KUKA KRL program: bl_1.src

&ACCESS RVP
&REL 1
&PARAM TEMPLATE = C:\KRC\Roboter\Template\vorgabe
&PARAM EDITMASK = *
DEF group15cm ( )


;FOLD INI
;FOLD BASISTECH INI
GLOBAL INTERRUPT DECL 3 WHEN $STOPMESS==TRUE DO IR_STOPM ( )
INTERRUPT ON 3
BAS (#INITMOV,0 )
;ENDFOLD (BASISTECH INI)
;ENDFOLD (INI)

;FOLD STARTPOSITION - BASE IS 2, TOOL IS 6, SPEED IS 45%, POSITION IS A1 5,A2 -30,A3 100,A4 5,A5 -60,A6 -135,E1 0,E2 0,E3 0,E4 0
$BWDSTART = FALSE
PDAT_ACT = {VEL 45,ACC 100,APO_DIST 50}
FDAT_ACT = {TOOL_NO 6,BASE_NO 2,IPO_FRAME #BASE}
BAS (#PTP_PARAMS,45)
PTP  {A1 5,A2 -30,A3 100,A4 5,A5 -60,A6 -135,E1 0,E2 0,E3 0,E4 0}
;ENDFOLD

;FOLD LIN SPEED IS 0.5 m/sec, INTERPOLATION SETTINGS IN FOLD
$VEL.CP=0.5
$ADVANCE=3
;ENDFOLD

PTP{ E6POS: X 793.0310, Y -5.4900, Z -174.0150, A 0, B 90, C 0, E1 0, E2 0, E3 0, E4 0, S 'B 110' } C_PTP
LIN{ E6POS: X 793.0310, Y -5.4900, Z -174.0150, A 0, B 90, C 0, E1 0, E2 0, E3 0, E4 0 }
LIN{ E6POS: X 792.7476, Y -6.4490, Z -174.0150, A 0, B 90, C 0, E1 0, E2 0, E3 0, E4 0 } C_DIS
LIN{ E6POS: X 792.4642, Y -7.4080, Z -174.0150, A 0, B 90, C 0, E1 0, E2 0, E3 0, E4 0 } C_DIS
LIN{ E6POS: X 792.1808, Y -8.3670, Z -174.0150, A 0, B 90, C 0, E1 0, E2 0, E3 0, E4 0 } C_DIS
LIN{ E6POS: X 791.8974, Y -9.3260, Z -174.0150, A 0, B 90, C 0, E1 0, E2 0, E3 0, E4 0 } C_DIS
LIN{ E6POS: X 791.6139, Y -10.2850, Z -174.0150, A 0, B 90, C 0, E1 0, E2 0, E3 0, E4 0 } C_DIS
LIN{ E6POS: X 791.3305, Y -11.2440, Z -174.0150, A 0, B 90, C 0, E1 0, E2 0, E3 0, E4 0 } C_DIS
LIN{ E6POS: X 791.0471, Y -12.2030, Z -174.0150, A 0, B 90, C 0, E1 0, E2 0, E3 0, E4 0 } C_DIS
LIN{ E6POS: X 790.7637, Y -13.1620, Z -174.0150, A 0, B 90, C 0, E1 0, E2 0, E3 0, E4 0 } C_DIS
LIN{ E6POS: X 790.4803, Y -14.1210, Z -174.0150, A 0, B 90, C 0, E1 0, E2 0, E3 0, E4 0 } C_DIS
LIN{ E6POS: X 790.2681, Y -14.8387, Z -174.0150, A 0, B 90, C 0, E1 0, E2 0, E3 0, E4 0 } C_DIS
LIN{ E6POS: X 790.2681, Y -14.8387, Z -174.0150, A 0, B 90, C 0, E1 0, E2 0, E3 0, E4 0 } C_DIS
LIN{ E6POS: X 789.6733, Y -15.6426, Z -174.0150, A 0, B 90, C 0, E1 0, E2 0, E3 0, E4 0 } C_DIS
LIN{ E6POS: X 789.0784, Y -16.4464, Z -174.0150, A 0, B 90, C 0, E1 0, E2 0, E3 0, E4 0 } C_DIS
LIN{ E6POS: X 788.4835, Y -17.2502, Z -174.0150, A 0, B 90, C 0, E1 0, E2 0, E3 0, E4 0 } C_DIS
LIN{ E6POS: X 787.8887, Y -18.0540, Z -174.0150, A 0, B 90, C 0, E1 0, E2 0, E3 0, E4 0 } C_DIS
LIN{ E6POS: X 787.2938, Y -18.8579, Z -174.0150, A 0, B 90, C 0, E1 0, E2 0, E3 0, E4 0 } C_DIS
LIN{ E6POS: X 786.7884, Y -19.5408, Z -174.0150, A 0, B 90, C 0, E1 0, E2 0, E3 0, E4 0 } C_DIS
LIN{ E6POS: X 786.7884, Y -19.5408, Z -174.0150, A 0, B 90, C 0, E1 0, E2 0, E3 0, E4 0 } C_DIS
LIN{ E6POS: X 785.8349, Y -19.8419, Z -174.0150, A 0, B 90, C 0, E1 0, E2 0, E3 0, E4 0 } C_DIS
LIN{ E6POS: X 784.8813, Y -20.1431, Z -174.0150, A 0, B 90, C 0, E1 0, E2 0, E3 0, E4 0 } C_DIS
LIN{ E6POS: X 783.9277, Y -20.4443, Z -174.0150, A 0, B 90, C 0, E1 0, E2 0, E3 0, E4 0 } C_DIS
LIN{ E6POS: X 782.9742, Y -20.7455, Z -174.0150, A 0, B 90, C 0, E1 0, E2 0, E3 0, E4 0 } C_DIS
LIN{ E6POS: X 782.5387, Y -20.8830, Z -174.0150, A 0, B 90, C 0, E1 0, E2 0, E3 0, E4 0 } C_DIS
LIN{ E6POS: X 781.5488, Y -20.7411, Z -174.0150, A 0, B 90, C 0, E1 0, E2 0, E3 0, E4 0 } C_DIS
LIN{ E6POS: X 780.5590, Y -20.5992, Z -174.0150, A 0, B 90, C 0, E1 0, E2 0, E3 0, E4 0 } C_DIS
LIN{ E6POS: X 779.5691, Y -20.4573, Z -174.0150, A 0, B 90, C 0, E1 0, E2 0, E3 0, E4 0 } C_DIS
LIN{ E6POS: X 778.5792, Y -20.3154, Z -174.0150, A 0, B 90, C 0, E1 0, E2 0, E3 0, E4 0 } C_DIS
LIN{ E6POS: X 777.5893, Y -20.1735, Z -174.0150, A 0, B 90, C 0, E1 0, E2 0, E3 0, E4 0 } C_DIS
LIN{ E6POS: X 777.4677, Y -20.1560, Z -174.0150, A 0, B 90, C 0, E1 0, E2 0, E3 0, E4 0 } C_DIS
LIN{ E6POS: X 777.4677, Y -20.1560, Z -174.0150, A 0, B 90, C 0, E1 0, E2 0, E3 0, E4 0 } C_DIS
LIN{ E6POS: X 776.4984, Y -19.9101, Z -174.0150, A 0, B 90, C 0, E1 0, E2 0, E3 0, E4 0 } C_DIS
LIN{ E6POS: X 775.5291, Y -19.6643, Z -174.0150, A 0, B 90, C 0, E1 0, E2 0, E3 0, E4 0 } C_DIS
LIN{ E6POS: X 774.5598, Y -19.4184, Z -174.0150, A 0, B 90, C 0, E1 0, E2 0, E3 0, E4 0 } C_DIS
LIN{ E6POS: X 773.5905, Y -19.1725, Z -174.0150, A 0, B 90, C 0, E1 0, E2 0, E3 0, E4 0 } C_DIS
LIN{ E6POS: X 772.6212, Y -18.9266, Z -174.0150, A 0, B 90, C 0, E1 0, E2 0, E3 0, E4 0 } C_DIS
LIN{ E6POS: X 771.6519, Y -18.6807, Z -174.0150, A 0, B 90, C 0, E1 0, E2 0, E3 0, E4 0 } C_DIS
LIN{ E6POS: X 771.5220, Y -18.6477, Z -174.0150, A 0, B 90, C 0, E1 0, E2 0, E3 0, E4 0 } C_DIS
LIN{ E6POS: X 771.5220, Y -18.6477, Z -174.0150, A 0, B 90, C 0, E1 0, E2 0, E3 0, E4 0 } C_DIS
LIN{ E6POS: X 770.5324, Y -18.5039, Z -174.0150, A 0, B 90, C 0, E1 0, E2 0, E3 0, E4 0 } C_DIS
LIN{ E6POS: X 769.5428, Y -18.3600, Z -174.0150, A 0, B 90, C 0, E1 0, E2 0, E3 0, E4 0 } C_DIS
LIN{ E6POS: X 768.5532, Y -18.2161, Z -174.0150, A 0, B 90, C 0, E1 0, E2 0, E3 0, E4 0 } C_DIS
LIN{ E6POS: X 767.5636, Y -18.0723, Z -174.0150, A 0, B 90, C 0, E1 0, E2 0, E3 0, E4 0 } C_DIS
LIN{ E6POS: X 766.5740, Y -17.9284, Z -174.0150, A 0, B 90, C 0, E1 0, E2 0, E3 0, E4 0 } C_DIS
LIN{ E6POS: X 765.5844, Y -17.7845, Z -174.0150, A 0, B 90, C 0, E1 0, E2 0, E3 0, E4 0 } C_DIS
LIN{ E6POS: X 764.6502, Y -17.6487, Z -174.0150, A 0, B 90, C 0, E1 0, E2 0, E3 0, E4 0 } C_DIS
LIN{ E6POS: X 764.6502, Y -17.6487, Z -174.0150, A 0, B 90, C 0, E1 0, E2 0, E3 0, E4 0 } C_DIS
LIN{ E6POS: X 763.6529, Y -17.5756, Z -174.0150, A 0, B 90, C 0, E1 0, E2 0, E3 0, E4 0 } C_DIS
LIN{ E6POS: X 762.6555, Y -17.5025, Z -174.0150, A 0, B 90, C 0, E1 0, E2 0, E3 0, E4 0 } C_DIS
LIN{ E6POS: X 761.6582, Y -17.4294, Z -174.0150, A 0, B 90, C 0, E1 0, E2 0, E3 0, E4 0 } C_DIS
LIN{ E6POS: X 760.6609, Y -17.3562, Z -174.0150, A 0, B 90, C 0, E1 0, E2 0, E3 0, E4 0 } C_DIS
LIN{ E6POS: X 759.6636, Y -17.2831, Z -174.0150, A 0, B 90, C 0, E1 0, E2 0, E3 0, E4 0 } C_DIS
LIN{ E6POS: X 758.6662, Y -17.2100, Z -174.0150, A 0, B 90, C 0, E1 0, E2 0, E3 0, E4 0 } C_DIS
LIN{ E6POS: X 757.6689, Y -17.1369, Z -174.0150, A 0, B 90, C 0, E1 0, E2 0, E3 0, E4 0 } C_DIS
LIN{ E6POS: X 757.5979, Y -17.1316, Z -174.0150, A 0, B 90, C 0, E1 0, E2 0, E3 0, E4 0 } C_DIS
LIN{ E6POS: X 757.5979, Y -17.1316, Z -174.0150, A 0, B 90, C 0, E1 0, E2 0, E3 0, E4 0 } C_DIS
LIN{ E6POS: X 756.5980, Y -17.1225, Z -174.0150, A 0, B 90, C 0, E1 0, E2 0, E3 0, E4 0 } C_DIS
LIN{ E6POS: X 755.5980, Y -17.1134, Z -174.0150, A 0, B 90, C 0, E1 0, E2 0, E3 0, E4 0 } C_DIS
LIN{ E6POS: X 754.5981, Y -17.1043, Z -174.0150, A 0, B 90, C 0, E1 0, E2 0, E3 0, E4 0 } C_DIS
LIN{ E6POS: X 753.5981, Y -17.0952, Z -174.0150, A 0, B 90, C 0, E1 0, E2 0, E3 0, E4 0 } C_DIS
LIN{ E6POS: X 752.5981, Y -17.0860, Z -174.0150, A 0, B 90, C 0, E1 0, E2 0, E3 0, E4 0 } C_DIS
LIN{ E6POS: X 751.5982, Y -17.0769, Z -174.0150, A 0, B 90, C 0, E1 0, E2 0, E3 0, E4 0 } C_DIS
LIN{ E6POS: X 751.1080, Y -17.0724, Z -174.0150, A 0, B 90, C 0, E1 0, E2 0, E3 0, E4 0 } C_DIS
LIN{ E6POS: X 751.1080, Y -17.0724, Z -174.0150, A 0, B 90, C 0, E1 0, E2 0, E3 0, E4 0 } C_DIS
LIN{ E6POS: X 750.1105, Y -17.1440, Z -174.0150, A 0, B 90, C 0, E1 0, E2 0, E3 0, E4 0 } C_DIS
LIN{ E6POS: X 749.1131, Y -17.2155, Z -174.0150, A 0, B 90, C 0, E1 0, E2 0, E3 0, E4 0 } C_DIS
LIN{ E6POS: X 748.1157, Y -17.2870, Z -174.0150, A 0, B 90, C 0, E1 0, E2 0, E3 0, E4 0 } C_DIS
LIN{ E6POS: X 747.1182, Y -17.3586, Z -174.0150, A 0, B 90, C 0, E1 0, E2 0, E3 0, E4 0 } C_DIS
LIN{ E6POS: X 746.1208, Y -17.4301, Z -174.0150, A 0, B 90, C 0, E1 0, E2 0, E3 0, E4 0 } C_DIS
LIN{ E6POS: X 745.9267, Y -17.4440, Z -174.0150, A 0, B 90, C 0, E1 0, E2 0, E3 0, E4 0 } C_DIS
LIN{ E6POS: X 745.9267, Y -17.4440, Z -174.0150, A 0, B 90, C 0, E1 0, E2 0, E3 0, E4 0 } C_DIS
LIN{ E6POS: X 744.9564, Y -17.6858, Z -174.0150, A 0, B 90, C 0, E1 0, E2 0, E3 0, E4 0 } C_DIS
LIN{ E6POS: X 743.9861, Y -17.9276, Z -174.0150, A 0, B 90, C 0, E1 0, E2 0, E3 0, E4 0 } C_DIS
LIN{ E6POS: X 743.0157, Y -18.1693, Z -174.0150, A 0, B 90, C 0, E1 0, E2 0, E3 0, E4 0 } C_DIS
LIN{ E6POS: X 742.7996, Y -18.2232, Z -174.0150, A 0, B 90, C 0, E1 0, E2 0, E3 0, E4 0 } C_DIS
LIN{ E6POS: X 742.7996, Y -18.2232, Z -174.0150, A 0, B 90, C 0, E1 0, E2 0, E3 0, E4 0 } C_DIS
LIN{ E6POS: X 742.1156, Y -18.9526, Z -174.0150, A 0, B 90, C 0, E1 0, E2 0, E3 0, E4 0 } C_DIS
LIN{ E6POS: X 741.7327, Y -19.3609, Z -174.0150, A 0, B 90, C 0, E1 0, E2 0, E3 0, E4 0 } C_DIS
LIN{ E6POS: X 741.7327, Y -19.3609, Z -174.0150, A 0, B 90, C 0, E1 0, E2 0, E3 0, E4 0 } C_DIS
LIN{ E6POS: X 741.7327, Y -19.3609, Z -174.0150, A 0, B 90, C 0, E1 0, E2 0, E3 0, E4 0 } C_DIS
LIN{ E6POS: X 742.3016, Y -20.1832, Z -174.0150, A 0, B 90, C 0, E1 0, E2 0, E3 0, E4 0 } C_DIS
LIN{ E6POS: X 742.7345, Y -20.8088, Z -174.0150, A 0, B 90, C 0, E1 0, E2 0, E3 0, E4 0 } C_DIS
LIN{ E6POS: X 742.7345, Y -20.8088, Z -174.0150, A 0, B 90, C 0, E1 0, E2 0, E3 0, E4 0 } C_DIS
LIN{ E6POS: X 743.6084, Y -21.2949, Z -174.0150, A 0, B 90, C 0, E1 0, E2 0, E3 0, E4 0 } C_DIS
LIN{ E6POS: X 744.4823, Y -21.7810, Z -174.0150, A 0, B 90, C 0, E1 0, E2 0, E3 0, E4 0 } C_DIS
LIN{ E6POS: X 745.3563, Y -22.2671, Z -174.0150, A 0, B 90, C 0, E1 0, E2 0, E3 0, E4 0 } C_DIS
LIN{ E6POS: X 745.8115, Y -22.5203, Z -174.0150, A 0, B 90, C 0, E1 0, E2 0, E3 0, E4 0 } C_DIS
LIN{ E6POS: X 745.8115, Y -22.5203, Z -174.0150, A 0, B 90, C 0, E1 0, E2 0, E3 0, E4 0 } C_DIS
LIN{ E6POS: X 746.7484, Y -22.8698, Z -174.0150, A 0, B 90, C 0, E1 0, E2 0, E3 0, E4 0 } C_DIS
LIN{ E6POS: X 747.6853, Y -23.2194, Z -174.0150, A 0, B 90, C 0, E1 0, E2 0, E3 0, E4 0 } C_DIS
LIN{ E6POS: X 748.6222, Y -23.5690, Z -174.0150, A 0, B 90, C 0, E1 0, E2 0, E3 0, E4 0 } C_DIS
LIN{ E6POS: X 749.5592, Y -23.9186, Z -174.0150, A 0, B 90, C 0, E1 0, E2 0, E3 0, E4 0 } C_DIS
LIN{ E6POS: X 750.4961, Y -24.2681, Z -174.0150, A 0, B 90, C 0, E1 0, E2 0, E3 0, E4 0 } C_DIS
LIN{ E6POS: X 750.9726, Y -24.4459, Z -174.0150, A 0, B 90, C 0, E1 0, E2 0, E3 0, E4 0 } C_DIS
LIN{ E6POS: X 750.9726, Y -24.4459, Z -174.0150, A 0, B 90, C 0, E1 0, E2 0, E3 0, E4 0 } C_DIS
LIN{ E6POS: X 751.9333, Y -24.7235, Z -174.0150, A 0, B 90, C 0, E1 0, E2 0, E3 0, E4 0 } C_DIS
LIN{ E6POS: X 752.8940, Y -25.0011, Z -174.0150, A 0, B 90, C 0, E1 0, E2 0, E3 0, E4 0 } C_DIS
LIN{ E6POS: X 753.8547, Y -25.2787, Z -174.0150, A 0, B 90, C 0, E1 0, E2 0, E3 0, E4 0 } C_DIS
LIN{ E6POS: X 754.8154, Y -25.5563, Z -174.0150, A 0, B 90, C 0, E1 0, E2 0, E3 0, E4 0 } C_DIS
LIN{ E6POS: X 755.7761, Y -25.8339, Z -174.0150, A 0, B 90, C 0, E1 0, E2 0, E3 0, E4 0 } C_DIS
LIN{ E6POS: X 756.7368, Y -26.1115, Z -174.0150, A 0, B 90, C 0, E1 0, E2 0, E3 0, E4 0 } C_DIS
LIN{ E6POS: X 757.4643, Y -26.3217, Z -174.0150, A 0, B 90, C 0, E1 0, E2 0, E3 0, E4 0 } C_DIS
LIN{ E6POS: X 757.4643, Y -26.3217, Z -174.0150, A 0, B 90, C 0, E1 0, E2 0, E3 0, E4 0 } C_DIS
LIN{ E6POS: X 758.4408, Y -26.5375, Z -174.0150, A 0, B 90, C 0, E1 0, E2 0, E3 0, E4 0 } C_DIS
LIN{ E6POS: X 759.4172, Y -26.7532, Z -174.0150, A 0, B 90, C 0, E1 0, E2 0, E3 0, E4 0 } C_DIS
LIN{ E6POS: X 760.3937, Y -26.9690, Z -174.0150, A 0, B 90, C 0, E1 0, E2 0, E3 0, E4 0 } C_DIS
LIN{ E6POS: X 761.3701, Y -27.1847, Z -174.0150, A 0, B 90, C 0, E1 0, E2 0, E3 0, E4 0 } C_DIS
LIN{ E6POS: X 762.3466, Y -27.4005, Z -174.0150, A 0, B 90, C 0, E1 0, E2 0, E3 0, E4 0 } C_DIS
LIN{ E6POS: X 763.3230, Y -27.6162, Z -174.0150, A 0, B 90, C 0, E1 0, E2 0, E3 0, E4 0 } C_DIS
LIN{ E6POS: X 764.2995, Y -27.8320, Z -174.0150, A 0, B 90, C 0, E1 0, E2 0, E3 0, E4 0 } C_DIS
LIN{ E6POS: X 764.5341, Y -27.8838, Z -174.0150, A 0, B 90, C 0, E1 0, E2 0, E3 0, E4 0 } C_DIS
LIN{ E6POS: X 764.5341, Y -27.8838, Z -174.0150, A 0, B 90, C 0, E1 0, E2 0, E3 0, E4 0 } C_DIS
LIN{ E6POS: X 765.5242, Y -28.0248, Z -174.0150, A 0, B 90, C 0, E1 0, E2 0, E3 0, E4 0 } C_DIS
LIN{ E6POS: X 766.5142, Y -28.1657, Z -174.0150, A 0, B 90, C 0, E1 0, E2 0, E3 0, E4 0 } C_DIS
LIN{ E6POS: X 767.5042, Y -28.3066, Z -174.0150, A 0, B 90, C 0, E1 0, E2 0, E3 0, E4 0 } C_DIS
LIN{ E6POS: X 768.4942, Y -28.4476, Z -174.0150, A 0, B 90, C 0, E1 0, E2 0, E3 0, E4 0 } C_DIS
LIN{ E6POS: X 769.4842, Y -28.5885, Z -174.0150, A 0, B 90, C 0, E1 0, E2 0, E3 0, E4 0 } C_DIS
LIN{ E6POS: X 770.4743, Y -28.7294, Z -174.0150, A 0, B 90, C 0, E1 0, E2 0, E3 0, E4 0 } C_DIS
LIN{ E6POS: X 771.4301, Y -28.8655, Z -174.0150, A 0, B 90, C 0, E1 0, E2 0, E3 0, E4 0 } C_DIS
LIN{ E6POS: X 771.4301, Y -28.8655, Z -174.0150, A 0, B 90, C 0, E1 0, E2 0, E3 0, E4 0 } C_DIS
LIN{ E6POS: X 772.4299, Y -28.8885, Z -174.0150, A 0, B 90, C 0, E1 0, E2 0, E3 0, E4 0 } C_DIS
LIN{ E6POS: X 773.4296, Y -28.9114, Z -174.0150, A 0, B 90, C 0, E1 0, E2 0, E3 0, E4 0 } C_DIS
LIN{ E6POS: X 774.4294, Y -28.9344, Z -174.0150, A 0, B 90, C 0, E1 0, E2 0, E3 0, E4 0 } C_DIS
LIN{ E6POS: X 775.4291, Y -28.9574, Z -174.0150, A 0, B 90, C 0, E1 0, E2 0, E3 0, E4 0 } C_DIS
LIN{ E6POS: X 776.4288, Y -28.9803, Z -174.0150, A 0, B 90, C 0, E1 0, E2 0, E3 0, E4 0 } C_DIS
LIN{ E6POS: X 777.3989, Y -29.0026, Z -174.0150, A 0, B 90, C 0, E1 0, E2 0, E3 0, E4 0 } C_DIS
LIN{ E6POS: X 777.3989, Y -29.0026, Z -174.0150, A 0, B 90, C 0, E1 0, E2 0, E3 0, E4 0 } C_DIS
LIN{ E6POS: X 778.3804, Y -29.1940, Z -174.0150, A 0, B 90, C 0, E1 0, E2 0, E3 0, E4 0 } C_DIS
LIN{ E6POS: X 779.3620, Y -29.3854, Z -174.0150, A 0, B 90, C 0, E1 0, E2 0, E3 0, E4 0 } C_DIS
LIN{ E6POS: X 780.3435, Y -29.5769, Z -174.0150, A 0, B 90, C 0, E1 0, E2 0, E3 0, E4 0 } C_DIS
LIN{ E6POS: X 781.3250, Y -29.7683, Z -174.0150, A 0, B 90, C 0, E1 0, E2 0, E3 0, E4 0 } C_DIS
LIN{ E6POS: X 782.0838, Y -29.9163, Z -174.0150, A 0, B 90, C 0, E1 0, E2 0, E3 0, E4 0 } C_DIS
LIN{ E6POS: X 782.0838, Y -29.9163, Z -174.0150, A 0, B 90, C 0, E1 0, E2 0, E3 0, E4 0 } C_DIS
LIN{ E6POS: X 782.7607, Y -30.6523, Z -174.0150, A 0, B 90, C 0, E1 0, E2 0, E3 0, E4 0 } C_DIS
LIN{ E6POS: X 783.4376, Y -31.3884, Z -174.0150, A 0, B 90, C 0, E1 0, E2 0, E3 0, E4 0 } C_DIS
LIN{ E6POS: X 784.1145, Y -32.1244, Z -174.0150, A 0, B 90, C 0, E1 0, E2 0, E3 0, E4 0 } C_DIS
LIN{ E6POS: X 784.7914, Y -32.8605, Z -174.0150, A 0, B 90, C 0, E1 0, E2 0, E3 0, E4 0 } C_DIS
LIN{ E6POS: X 785.1281, Y -33.2266, Z -174.0150, A 0, B 90, C 0, E1 0, E2 0, E3 0, E4 0 } C_DIS
LIN{ E6POS: X 785.1281, Y -33.2266, Z -174.0150, A 0, B 90, C 0, E1 0, E2 0, E3 0, E4 0 } C_DIS
LIN{ E6POS: X 785.2695, Y -34.2166, Z -174.0150, A 0, B 90, C 0, E1 0, E2 0, E3 0, E4 0 } C_DIS
LIN{ E6POS: X 785.4109, Y -35.2065, Z -174.0150, A 0, B 90, C 0, E1 0, E2 0, E3 0, E4 0 } C_DIS
LIN{ E6POS: X 785.5523, Y -36.1965, Z -174.0150, A 0, B 90, C 0, E1 0, E2 0, E3 0, E4 0 } C_DIS
LIN{ E6POS: X 785.6937, Y -37.1864, Z -174.0150, A 0, B 90, C 0, E1 0, E2 0, E3 0, E4 0 } C_DIS
LIN{ E6POS: X 785.8351, Y -38.1764, Z -174.0150, A 0, B 90, C 0, E1 0, E2 0, E3 0, E4 0 } C_DIS
LIN{ E6POS: X 785.9765, Y -39.1663, Z -174.0150, A 0, B 90, C 0, E1 0, E2 0, E3 0, E4 0 } C_DIS
LIN{ E6POS: X 786.1179, Y -40.1563, Z -174.0150, A 0, B 90, C 0, E1 0, E2 0, E3 0, E4 0 } C_DIS
LIN{ E6POS: X 786.1747, Y -40.5536, Z -174.0150, A 0, B 90, C 0, E1 0, E2 0, E3 0, E4 0 } C_DIS
LIN{ E6POS: X 786.1747, Y -40.5536, Z -174.0150, A 0, B 90, C 0, E1 0, E2 0, E3 0, E4 0 } C_DIS
LIN{ E6POS: X 786.0743, Y -41.5485, Z -174.0150, A 0, B 90, C 0, E1 0, E2 0, E3 0, E4 0 } C_DIS
LIN{ E6POS: X 785.9740, Y -42.5435, Z -174.0150, A 0, B 90, C 0, E1 0, E2 0, E3 0, E4 0 } C_DIS
LIN{ E6POS: X 785.8737, Y -43.5384, Z -174.0150, A 0, B 90, C 0, E1 0, E2 0, E3 0, E4 0 } C_DIS
LIN{ E6POS: X 785.7734, Y -44.5334, Z -174.0150, A 0, B 90, C 0, E1 0, E2 0, E3 0, E4 0 } C_DIS
LIN{ E6POS: X 785.6731, Y -45.5283, Z -174.0150, A 0, B 90, C 0, E1 0, E2 0, E3 0, E4 0 } C_DIS
LIN{ E6POS: X 785.5728, Y -46.5233, Z -174.0150, A 0, B 90, C 0, E1 0, E2 0, E3 0, E4 0 } C_DIS
LIN{ E6POS: X 785.4725, Y -47.5183, Z -174.0150, A 0, B 90, C 0, E1 0, E2 0, E3 0, E4 0 } C_DIS
LIN{ E6POS: X 785.3721, Y -48.5132, Z -174.0150, A 0, B 90, C 0, E1 0, E2 0, E3 0, E4 0 } C_DIS
LIN{ E6POS: X 785.2718, Y -49.5082, Z -174.0150, A 0, B 90, C 0, E1 0, E2 0, E3 0, E4 0 } C_DIS
LIN{ E6POS: X 785.1715, Y -50.5031, Z -174.0150, A 0, B 90, C 0, E1 0, E2 0, E3 0, E4 0 } C_DIS
LIN{ E6POS: X 785.0712, Y -51.4981, Z -174.0150, A 0, B 90, C 0, E1 0, E2 0, E3 0, E4 0 } C_DIS
LIN{ E6POS: X 784.9709, Y -52.4930, Z -174.0150, A 0, B 90, C 0, E1 0, E2 0, E3 0, E4 0 } C_DIS
LIN{ E6POS: X 784.8706, Y -53.4880, Z -174.0150, A 0, B 90, C 0, E1 0, E2 0, E3 0, E4 0 } C_DIS
LIN{ E6POS: X 784.8675, Y -53.5185, Z -174.0150, A 0, B 90, C 0, E1 0, E2 0, E3 0, E4 0 } C_DIS
LIN{ E6POS: X 784.8675, Y -53.5185, Z -174.0150, A 0, B 90, C 0, E1 0, E2 0, E3 0, E4 0 } C_DIS
LIN{ E6POS: X 784.6915, Y -54.5029, Z -174.0150, A 0, B 90, C 0, E1 0, E2 0, E3 0, E4 0 } C_DIS
LIN{ E6POS: X 784.5156, Y -55.4873, Z -174.0150, A 0, B 90, C 0, E1 0, E2 0, E3 0, E4 0 } C_DIS
LIN{ E6POS: X 784.3396, Y -56.4717, Z -174.0150, A 0, B 90, C 0, E1 0, E2 0, E3 0, E4 0 } C_DIS
LIN{ E6POS: X 784.1637, Y -57.4560, Z -174.0150, A 0, B 90, C 0, E1 0, E2 0, E3 0, E4 0 } C_DIS
LIN{ E6POS: X 783.9877, Y -58.4404, Z -174.0150, A 0, B 90, C 0, E1 0, E2 0, E3 0, E4 0 } C_DIS
LIN{ E6POS: X 783.8118, Y -59.4248, Z -174.0150, A 0, B 90, C 0, E1 0, E2 0, E3 0, E4 0 } C_DIS
LIN{ E6POS: X 783.6358, Y -60.4092, Z -174.0150, A 0, B 90, C 0, E1 0, E2 0, E3 0, E4 0 } C_DIS
LIN{ E6POS: X 783.4599, Y -61.3936, Z -174.0150, A 0, B 90, C 0, E1 0, E2 0, E3 0, E4 0 } C_DIS
LIN{ E6POS: X 783.2839, Y -62.3780, Z -174.0150, A 0, B 90, C 0, E1 0, E2 0, E3 0, E4 0 } C_DIS
LIN{ E6POS: X 783.1080, Y -63.3624, Z -174.0150, A 0, B 90, C 0, E1 0, E2 0, E3 0, E4 0 } C_DIS
LIN{ E6POS: X 782.9320, Y -64.3468, Z -174.0150, A 0, B 90, C 0, E1 0, E2 0, E3 0, E4 0 } C_DIS
LIN{ E6POS: X 782.7561, Y -65.3312, Z -174.0150, A 0, B 90, C 0, E1 0, E2 0, E3 0, E4 0 } C_DIS
LIN{ E6POS: X 782.5801, Y -66.3156, Z -174.0150, A 0, B 90, C 0, E1 0, E2 0, E3 0, E4 0 } C_DIS
LIN{ E6POS: X 782.4042, Y -67.3000, Z -174.0150, A 0, B 90, C 0, E1 0, E2 0, E3 0, E4 0 } C_DIS
LIN{ E6POS: X 782.2282, Y -68.2844, Z -174.0150, A 0, B 90, C 0, E1 0, E2 0, E3 0, E4 0 } C_DIS
LIN{ E6POS: X 782.0523, Y -69.2688, Z -174.0150, A 0, B 90, C 0, E1 0, E2 0, E3 0, E4 0 } C_DIS
LIN{ E6POS: X 781.8763, Y -70.2532, Z -174.0150, A 0, B 90, C 0, E1 0, E2 0, E3 0, E4 0 } C_DIS
LIN{ E6POS: X 781.7943, Y -70.7119, Z -174.0150, A 0, B 90, C 0, E1 0, E2 0, E3 0, E4 0 } C_DIS
LIN{ E6POS: X 781.7943, Y -70.7119, Z -174.0150, A 0, B 90, C 0, E1 0, E2 0, E3 0, E4 0 } C_DIS
LIN{ E6POS: X 781.5865, Y -71.6900, Z -174.0150, A 0, B 90, C 0, E1 0, E2 0, E3 0, E4 0 } C_DIS
LIN{ E6POS: X 781.3787, Y -72.6682, Z -174.0150, A 0, B 90, C 0, E1 0, E2 0, E3 0, E4 0 } C_DIS
LIN{ E6POS: X 781.1709, Y -73.6464, Z -174.0150, A 0, B 90, C 0, E1 0, E2 0, E3 0, E4 0 } C_DIS
LIN{ E6POS: X 780.9631, Y -74.6245, Z -174.0150, A 0, B 90, C 0, E1 0, E2 0, E3 0, E4 0 } C_DIS
LIN{ E6POS: X 780.7553, Y -75.6027, Z -174.0150, A 0, B 90, C 0, E1 0, E2 0, E3 0, E4 0 } C_DIS
LIN{ E6POS: X 780.5475, Y -76.5809, Z -174.0150, A 0, B 90, C 0, E1 0, E2 0, E3 0, E4 0 } C_DIS
LIN{ E6POS: X 780.3397, Y -77.5590, Z -174.0150, A 0, B 90, C 0, E1 0, E2 0, E3 0, E4 0 } C_DIS
LIN{ E6POS: X 780.1319, Y -78.5372, Z -174.0150, A 0, B 90, C 0, E1 0, E2 0, E3 0, E4 0 } C_DIS
LIN{ E6POS: X 779.9241, Y -79.5154, Z -174.0150, A 0, B 90, C 0, E1 0, E2 0, E3 0, E4 0 } C_DIS
LIN{ E6POS: X 779.7163, Y -80.4936, Z -174.0150, A 0, B 90, C 0, E1 0, E2 0, E3 0, E4 0 } C_DIS
LIN{ E6POS: X 779.5085, Y -81.4717, Z -174.0150, A 0, B 90, C 0, E1 0, E2 0, E3 0, E4 0 } C_DIS
LIN{ E6POS: X 779.3007, Y -82.4499, Z -174.0150, A 0, B 90, C 0, E1 0, E2 0, E3 0, E4 0 } C_DIS
LIN{ E6POS: X 779.0929, Y -83.4281, Z -174.0150, A 0, B 90, C 0, E1 0, E2 0, E3 0, E4 0 } C_DIS
LIN{ E6POS: X 778.8851, Y -84.4062, Z -174.0150, A 0, B 90, C 0, E1 0, E2 0, E3 0, E4 0 } C_DIS
LIN{ E6POS: X 778.6773, Y -85.3844, Z -174.0150, A 0, B 90, C 0, E1 0, E2 0, E3 0, E4 0 } C_DIS
LIN{ E6POS: X 778.4695, Y -86.3626, Z -174.0150, A 0, B 90, C 0, E1 0, E2 0, E3 0, E4 0 } C_DIS
LIN{ E6POS: X 778.2617, Y -87.3408, Z -174.0150, A 0, B 90, C 0, E1 0, E2 0, E3 0, E4 0 } C_DIS
LIN{ E6POS: X 778.0539, Y -88.3189, Z -174.0150, A 0, B 90, C 0, E1 0, E2 0, E3 0, E4 0 } C_DIS
LIN{ E6POS: X 777.8461, Y -89.2971, Z -174.0150, A 0, B 90, C 0, E1 0, E2 0, E3 0, E4 0 } C_DIS
LIN{ E6POS: X 777.6383, Y -90.2753, Z -174.0150, A 0, B 90, C 0, E1 0, E2 0, E3 0, E4 0 } C_DIS
LIN{ E6POS: X 777.5429, Y -90.7243, Z -174.0150, A 0, B 90, C 0, E1 0, E2 0, E3 0, E4 0 } C_DIS
LIN{ E6POS: X 777.5429, Y -90.7243, Z -174.0150, A 0, B 90, C 0, E1 0, E2 0, E3 0, E4 0 } C_DIS
LIN{ E6POS: X 777.3226, Y -91.6997, Z -174.0150, A 0, B 90, C 0, E1 0, E2 0, E3 0, E4 0 } C_DIS
LIN{ E6POS: X 777.1022, Y -92.6751, Z -174.0150, A 0, B 90, C 0, E1 0, E2 0, E3 0, E4 0 } C_DIS
LIN{ E6POS: X 776.8819, Y -93.6506, Z -174.0150, A 0, B 90, C 0, E1 0, E2 0, E3 0, E4 0 } C_DIS
LIN{ E6POS: X 776.6615, Y -94.6260, Z -174.0150, A 0, B 90, C 0, E1 0, E2 0, E3 0, E4 0 } C_DIS
LIN{ E6POS: X 776.4412, Y -95.6014, Z -174.0150, A 0, B 90, C 0, E1 0, E2 0, E3 0, E4 0 } C_DIS
LIN{ E6POS: X 776.2208, Y -96.5768, Z -174.0150, A 0, B 90, C 0, E1 0, E2 0, E3 0, E4 0 } C_DIS
LIN{ E6POS: X 776.0005, Y -97.5522, Z -174.0150, A 0, B 90, C 0, E1 0, E2 0, E3 0, E4 0 } C_DIS
LIN{ E6POS: X 775.7802, Y -98.5277, Z -174.0150, A 0, B 90, C 0, E1 0, E2 0, E3 0, E4 0 } C_DIS
LIN{ E6POS: X 775.5598, Y -99.5031, Z -174.0150, A 0, B 90, C 0, E1 0, E2 0, E3 0, E4 0 } C_DIS
LIN{ E6POS: X 775.3395, Y -100.4785, Z -174.0150, A 0, B 90, C 0, E1 0, E2 0, E3 0, E4 0 } C_DIS
LIN{ E6POS: X 775.1191, Y -101.4539, Z -174.0150, A 0, B 90, C 0, E1 0, E2 0, E3 0, E4 0 } C_DIS
LIN{ E6POS: X 774.8988, Y -102.4294, Z -174.0150, A 0, B 90, C 0, E1 0, E2 0, E3 0, E4 0 } C_DIS
LIN{ E6POS: X 774.6784, Y -103.4048, Z -174.0150, A 0, B 90, C 0, E1 0, E2 0, E3 0, E4 0 } C_DIS
LIN{ E6POS: X 774.4581, Y -104.3802, Z -174.0150, A 0, B 90, C 0, E1 0, E2 0, E3 0, E4 0 } C_DIS
LIN{ E6POS: X 774.2377, Y -105.3556, Z -174.0150, A 0, B 90, C 0, E1 0, E2 0, E3 0, E4 0 } C_DIS
LIN{ E6POS: X 774.0174, Y -106.3310, Z -174.0150, A 0, B 90, C 0, E1 0, E2 0, E3 0, E4 0 } C_DIS
LIN{ E6POS: X 773.7970, Y -107.3065, Z -174.0150, A 0, B 90, C 0, E1 0, E2 0, E3 0, E4 0 } C_DIS
LIN{ E6POS: X 773.5767, Y -108.2819, Z -174.0150, A 0, B 90, C 0, E1 0, E2 0, E3 0, E4 0 } C_DIS
LIN{ E6POS: X 773.3564, Y -109.2573, Z -174.0150, A 0, B 90, C 0, E1 0, E2 0, E3 0, E4 0 } C_DIS
LIN{ E6POS: X 773.1360, Y -110.2327, Z -174.0150, A 0, B 90, C 0, E1 0, E2 0, E3 0, E4 0 } C_DIS
LIN{ E6POS: X 772.9157, Y -111.2082, Z -174.0150, A 0, B 90, C 0, E1 0, E2 0, E3 0, E4 0 } C_DIS
LIN{ E6POS: X 772.7038, Y -112.1462, Z -174.0150, A 0, B 90, C 0, E1 0, E2 0, E3 0, E4 0 } C_DIS
LIN{ E6POS: X 772.7038, Y -112.1462, Z -174.0150, A 0, B 90, C 0, E1 0, E2 0, E3 0, E4 0 } C_DIS
LIN{ E6POS: X 772.0412, Y -111.3972, Z -174.0150, A 0, B 90, C 0, E1 0, E2 0, E3 0, E4 0 } C_DIS
LIN{ E6POS: X 771.3787, Y -110.6481, Z -174.0150, A 0, B 90, C 0, E1 0, E2 0, E3 0, E4 0 } C_DIS
LIN{ E6POS: X 770.7162, Y -109.8991, Z -174.0150, A 0, B 90, C 0, E1 0, E2 0, E3 0, E4 0 } C_DIS
LIN{ E6POS: X 770.0537, Y -109.1500, Z -174.0150, A 0, B 90, C 0, E1 0, E2 0, E3 0, E4 0 } C_DIS
LIN{ E6POS: X 770.0315, Y -109.1250, Z -174.0150, A 0, B 90, C 0, E1 0, E2 0, E3 0, E4 0 } C_DIS
LIN{ E6POS: X 770.0315, Y -109.1250, Z -174.0150, A 0, B 90, C 0, E1 0, E2 0, E3 0, E4 0 } C_DIS
LIN{ E6POS: X 769.2922, Y -108.4516, Z -174.0150, A 0, B 90, C 0, E1 0, E2 0, E3 0, E4 0 } C_DIS
LIN{ E6POS: X 768.5529, Y -107.7782, Z -174.0150, A 0, B 90, C 0, E1 0, E2 0, E3 0, E4 0 } C_DIS
LIN{ E6POS: X 767.8136, Y -107.1049, Z -174.0150, A 0, B 90, C 0, E1 0, E2 0, E3 0, E4 0 } C_DIS
LIN{ E6POS: X 767.0743, Y -106.4315, Z -174.0150, A 0, B 90, C 0, E1 0, E2 0, E3 0, E4 0 } C_DIS
LIN{ E6POS: X 766.6042, Y -106.0034, Z -174.0150, A 0, B 90, C 0, E1 0, E2 0, E3 0, E4 0 } C_DIS
LIN{ E6POS: X 765.7746, Y -105.4449, Z -174.0150, A 0, B 90, C 0, E1 0, E2 0, E3 0, E4 0 } C_DIS
LIN{ E6POS: X 764.9451, Y -104.8865, Z -174.0150, A 0, B 90, C 0, E1 0, E2 0, E3 0, E4 0 } C_DIS
LIN{ E6POS: X 764.1156, Y -104.3281, Z -174.0150, A 0, B 90, C 0, E1 0, E2 0, E3 0, E4 0 } C_DIS
LIN{ E6POS: X 763.2860, Y -103.7696, Z -174.0150, A 0, B 90, C 0, E1 0, E2 0, E3 0, E4 0 } C_DIS
LIN{ E6POS: X 762.4565, Y -103.2112, Z -174.0150, A 0, B 90, C 0, E1 0, E2 0, E3 0, E4 0 } C_DIS
LIN{ E6POS: X 761.6679, Y -102.6803, Z -174.0150, A 0, B 90, C 0, E1 0, E2 0, E3 0, E4 0 } C_DIS
LIN{ E6POS: X 761.6679, Y -102.6803, Z -174.0150, A 0, B 90, C 0, E1 0, E2 0, E3 0, E4 0 } C_DIS
LIN{ E6POS: X 760.7746, Y -102.2308, Z -174.0150, A 0, B 90, C 0, E1 0, E2 0, E3 0, E4 0 } C_DIS
LIN{ E6POS: X 759.8814, Y -101.7812, Z -174.0150, A 0, B 90, C 0, E1 0, E2 0, E3 0, E4 0 } C_DIS
LIN{ E6POS: X 758.9881, Y -101.3317, Z -174.0150, A 0, B 90, C 0, E1 0, E2 0, E3 0, E4 0 } C_DIS
LIN{ E6POS: X 758.0949, Y -100.8821, Z -174.0150, A 0, B 90, C 0, E1 0, E2 0, E3 0, E4 0 } C_DIS
LIN{ E6POS: X 757.2016, Y -100.4326, Z -174.0150, A 0, B 90, C 0, E1 0, E2 0, E3 0, E4 0 } C_DIS
LIN{ E6POS: X 756.3083, Y -99.9830, Z -174.0150, A 0, B 90, C 0, E1 0, E2 0, E3 0, E4 0 } C_DIS
LIN{ E6POS: X 755.4151, Y -99.5334, Z -174.0150, A 0, B 90, C 0, E1 0, E2 0, E3 0, E4 0 } C_DIS
LIN{ E6POS: X 754.5218, Y -99.0839, Z -174.0150, A 0, B 90, C 0, E1 0, E2 0, E3 0, E4 0 } C_DIS
LIN{ E6POS: X 754.4672, Y -99.0564, Z -174.0150, A 0, B 90, C 0, E1 0, E2 0, E3 0, E4 0 } C_DIS
LIN{ E6POS: X 754.4672, Y -99.0564, Z -174.0150, A 0, B 90, C 0, E1 0, E2 0, E3 0, E4 0 } C_DIS
LIN{ E6POS: X 753.5368, Y -98.6899, Z -174.0150, A 0, B 90, C 0, E1 0, E2 0, E3 0, E4 0 } C_DIS
LIN{ E6POS: X 752.6064, Y -98.3233, Z -174.0150, A 0, B 90, C 0, E1 0, E2 0, E3 0, E4 0 } C_DIS
LIN{ E6POS: X 751.6760, Y -97.9568, Z -174.0150, A 0, B 90, C 0, E1 0, E2 0, E3 0, E4 0 } C_DIS
LIN{ E6POS: X 750.7456, Y -97.5902, Z -174.0150, A 0, B 90, C 0, E1 0, E2 0, E3 0, E4 0 } C_DIS
LIN{ E6POS: X 749.8152, Y -97.2237, Z -174.0150, A 0, B 90, C 0, E1 0, E2 0, E3 0, E4 0 } C_DIS
LIN{ E6POS: X 748.8848, Y -96.8572, Z -174.0150, A 0, B 90, C 0, E1 0, E2 0, E3 0, E4 0 } C_DIS
LIN{ E6POS: X 747.9544, Y -96.4906, Z -174.0150, A 0, B 90, C 0, E1 0, E2 0, E3 0, E4 0 } C_DIS
LIN{ E6POS: X 747.0240, Y -96.1241, Z -174.0150, A 0, B 90, C 0, E1 0, E2 0, E3 0, E4 0 } C_DIS
LIN{ E6POS: X 746.0936, Y -95.7575, Z -174.0150, A 0, B 90, C 0, E1 0, E2 0, E3 0, E4 0 } C_DIS
LIN{ E6POS: X 745.1632, Y -95.3910, Z -174.0150, A 0, B 90, C 0, E1 0, E2 0, E3 0, E4 0 } C_DIS
LIN{ E6POS: X 744.2483, Y -95.0306, Z -174.0150, A 0, B 90, C 0, E1 0, E2 0, E3 0, E4 0 } C_DIS
LIN{ E6POS: X 744.2483, Y -95.0306, Z -174.0150, A 0, B 90, C 0, E1 0, E2 0, E3 0, E4 0 } C_DIS
LIN{ E6POS: X 743.3053, Y -94.6978, Z -174.0150, A 0, B 90, C 0, E1 0, E2 0, E3 0, E4 0 } C_DIS
LIN{ E6POS: X 742.3623, Y -94.3651, Z -174.0150, A 0, B 90, C 0, E1 0, E2 0, E3 0, E4 0 } C_DIS
LIN{ E6POS: X 741.4192, Y -94.0324, Z -174.0150, A 0, B 90, C 0, E1 0, E2 0, E3 0, E4 0 } C_DIS
LIN{ E6POS: X 740.4762, Y -93.6997, Z -174.0150, A 0, B 90, C 0, E1 0, E2 0, E3 0, E4 0 } C_DIS
LIN{ E6POS: X 739.5332, Y -93.3670, Z -174.0150, A 0, B 90, C 0, E1 0, E2 0, E3 0, E4 0 } C_DIS
LIN{ E6POS: X 738.5902, Y -93.0343, Z -174.0150, A 0, B 90, C 0, E1 0, E2 0, E3 0, E4 0 } C_DIS
LIN{ E6POS: X 737.6471, Y -92.7016, Z -174.0150, A 0, B 90, C 0, E1 0, E2 0, E3 0, E4 0 } C_DIS
LIN{ E6POS: X 736.7041, Y -92.3688, Z -174.0150, A 0, B 90, C 0, E1 0, E2 0, E3 0, E4 0 } C_DIS
LIN{ E6POS: X 735.7611, Y -92.0361, Z -174.0150, A 0, B 90, C 0, E1 0, E2 0, E3 0, E4 0 } C_DIS
LIN{ E6POS: X 734.8180, Y -91.7034, Z -174.0150, A 0, B 90, C 0, E1 0, E2 0, E3 0, E4 0 } C_DIS
LIN{ E6POS: X 733.8750, Y -91.3707, Z -174.0150, A 0, B 90, C 0, E1 0, E2 0, E3 0, E4 0 } C_DIS
LIN{ E6POS: X 732.9320, Y -91.0380, Z -174.0150, A 0, B 90, C 0, E1 0, E2 0, E3 0, E4 0 } C_DIS
LIN{ E6POS: X 732.7022, Y -90.9569, Z -174.0150, A 0, B 90, C 0, E1 0, E2 0, E3 0, E4 0 } C_DIS
LIN{ E6POS: X 732.7022, Y -90.9569, Z -174.0150, A 0, B 90, C 0, E1 0, E2 0, E3 0, E4 0 } C_DIS
LIN{ E6POS: X 731.7545, Y -90.6378, Z -174.0150, A 0, B 90, C 0, E1 0, E2 0, E3 0, E4 0 } C_DIS
LIN{ E6POS: X 730.8068, Y -90.3187, Z -174.0150, A 0, B 90, C 0, E1 0, E2 0, E3 0, E4 0 } C_DIS
LIN{ E6POS: X 729.8591, Y -89.9996, Z -174.0150, A 0, B 90, C 0, E1 0, E2 0, E3 0, E4 0 } C_DIS
LIN{ E6POS: X 728.9114, Y -89.6805, Z -174.0150, A 0, B 90, C 0, E1 0, E2 0, E3 0, E4 0 } C_DIS
LIN{ E6POS: X 727.9637, Y -89.3613, Z -174.0150, A 0, B 90, C 0, E1 0, E2 0, E3 0, E4 0 } C_DIS
LIN{ E6POS: X 727.0159, Y -89.0422, Z -174.0150, A 0, B 90, C 0, E1 0, E2 0, E3 0, E4 0 } C_DIS
LIN{ E6POS: X 726.0682, Y -88.7231, Z -174.0150, A 0, B 90, C 0, E1 0, E2 0, E3 0, E4 0 } C_DIS
LIN{ E6POS: X 725.1205, Y -88.4040, Z -174.0150, A 0, B 90, C 0, E1 0, E2 0, E3 0, E4 0 } C_DIS
LIN{ E6POS: X 724.1728, Y -88.0849, Z -174.0150, A 0, B 90, C 0, E1 0, E2 0, E3 0, E4 0 } C_DIS
LIN{ E6POS: X 723.2251, Y -87.7658, Z -174.0150, A 0, B 90, C 0, E1 0, E2 0, E3 0, E4 0 } C_DIS
LIN{ E6POS: X 722.2774, Y -87.4466, Z -174.0150, A 0, B 90, C 0, E1 0, E2 0, E3 0, E4 0 } C_DIS
LIN{ E6POS: X 721.5205, Y -87.1918, Z -174.0150, A 0, B 90, C 0, E1 0, E2 0, E3 0, E4 0 } C_DIS
LIN{ E6POS: X 721.5205, Y -87.1918, Z -174.0150, A 0, B 90, C 0, E1 0, E2 0, E3 0, E4 0 } C_DIS
LIN{ E6POS: X 720.5737, Y -86.8697, Z -174.0150, A 0, B 90, C 0, E1 0, E2 0, E3 0, E4 0 } C_DIS
LIN{ E6POS: X 719.6270, Y -86.5477, Z -174.0150, A 0, B 90, C 0, E1 0, E2 0, E3 0, E4 0 } C_DIS
LIN{ E6POS: X 718.6803, Y -86.2256, Z -174.0150, A 0, B 90, C 0, E1 0, E2 0, E3 0, E4 0 } C_DIS
LIN{ E6POS: X 717.7336, Y -85.9036, Z -174.0150, A 0, B 90, C 0, E1 0, E2 0, E3 0, E4 0 } C_DIS
LIN{ E6POS: X 716.7868, Y -85.5815, Z -174.0150, A 0, B 90, C 0, E1 0, E2 0, E3 0, E4 0 } C_DIS
LIN{ E6POS: X 715.8401, Y -85.2595, Z -174.0150, A 0, B 90, C 0, E1 0, E2 0, E3 0, E4 0 } C_DIS
LIN{ E6POS: X 714.8934, Y -84.9374, Z -174.0150, A 0, B 90, C 0, E1 0, E2 0, E3 0, E4 0 } C_DIS
LIN{ E6POS: X 713.9467, Y -84.6154, Z -174.0150, A 0, B 90, C 0, E1 0, E2 0, E3 0, E4 0 } C_DIS
LIN{ E6POS: X 713.0000, Y -84.2933, Z -174.0150, A 0, B 90, C 0, E1 0, E2 0, E3 0, E4 0 } C_DIS
LIN{ E6POS: X 712.3946, Y -84.0874, Z -174.0150, A 0, B 90, C 0, E1 0, E2 0, E3 0, E4 0 } C_DIS
LIN{ E6POS: X 712.3946, Y -84.0874, Z -174.0150, A 0, B 90, C 0, E1 0, E2 0, E3 0, E4 0 } C_DIS
LIN{ E6POS: X 711.4623, Y -83.7256, Z -174.0150, A 0, B 90, C 0, E1 0, E2 0, E3 0, E4 0 } C_DIS
LIN{ E6POS: X 710.5300, Y -83.3638, Z -174.0150, A 0, B 90, C 0, E1 0, E2 0, E3 0, E4 0 } C_DIS
LIN{ E6POS: X 709.5978, Y -83.0020, Z -174.0150, A 0, B 90, C 0, E1 0, E2 0, E3 0, E4 0 } C_DIS
LIN{ E6POS: X 708.6655, Y -82.6402, Z -174.0150, A 0, B 90, C 0, E1 0, E2 0, E3 0, E4 0 } C_DIS
LIN{ E6POS: X 707.7333, Y -82.2784, Z -174.0150, A 0, B 90, C 0, E1 0, E2 0, E3 0, E4 0 } C_DIS
LIN{ E6POS: X 707.0151, Y -81.9998, Z -174.0150, A 0, B 90, C 0, E1 0, E2 0, E3 0, E4 0 } C_DIS
LIN{ E6POS: X 707.0151, Y -81.9998, Z -174.0150, A 0, B 90, C 0, E1 0, E2 0, E3 0, E4 0 } C_DIS
LIN{ E6POS: X 706.1265, Y -81.5412, Z -174.0150, A 0, B 90, C 0, E1 0, E2 0, E3 0, E4 0 } C_DIS
LIN{ E6POS: X 705.2378, Y -81.0827, Z -174.0150, A 0, B 90, C 0, E1 0, E2 0, E3 0, E4 0 } C_DIS
LIN{ E6POS: X 704.4456, Y -80.6739, Z -174.0150, A 0, B 90, C 0, E1 0, E2 0, E3 0, E4 0 } C_DIS
LIN{ E6POS: X 704.4456, Y -80.6739, Z -174.0150, A 0, B 90, C 0, E1 0, E2 0, E3 0, E4 0 } C_DIS
LIN{ E6POS: X 704.0366, Y -79.7614, Z -174.0150, A 0, B 90, C 0, E1 0, E2 0, E3 0, E4 0 } C_DIS
LIN{ E6POS: X 703.9111, Y -79.4815, Z -174.0150, A 0, B 90, C 0, E1 0, E2 0, E3 0, E4 0 } C_DIS
LIN{ E6POS: X 703.9111, Y -79.4815, Z -174.0150, A 0, B 90, C 0, E1 0, E2 0, E3 0, E4 0 } C_DIS
LIN{ E6POS: X 703.9111, Y -79.4815, Z -174.0150, A 0, B 90, C 0, E1 0, E2 0, E3 0, E4 0 } C_DIS
LIN{ E6POS: X 704.2075, Y -78.5265, Z -174.0150, A 0, B 90, C 0, E1 0, E2 0, E3 0, E4 0 } C_DIS
LIN{ E6POS: X 704.4565, Y -77.7241, Z -174.0150, A 0, B 90, C 0, E1 0, E2 0, E3 0, E4 0 } C_DIS
LIN{ E6POS: X 704.4565, Y -77.7241, Z -174.0150, A 0, B 90, C 0, E1 0, E2 0, E3 0, E4 0 } C_DIS
LIN{ E6POS: X 704.7433, Y -76.7661, Z -174.0150, A 0, B 90, C 0, E1 0, E2 0, E3 0, E4 0 } C_DIS
LIN{ E6POS: X 704.9185, Y -76.1807, Z -174.0150, A 0, B 90, C 0, E1 0, E2 0, E3 0, E4 0 } C_DIS
LIN{ E6POS: X 704.9185, Y -76.1807, Z -174.0150, A 0, B 90, C 0, E1 0, E2 0, E3 0, E4 0 } C_DIS
LIN{ E6POS: X 705.2116, Y -75.2246, Z -174.0150, A 0, B 90, C 0, E1 0, E2 0, E3 0, E4 0 } C_DIS
LIN{ E6POS: X 705.3758, Y -74.6888, Z -174.0150, A 0, B 90, C 0, E1 0, E2 0, E3 0, E4 0 } C_DIS
LIN{ E6POS: X 705.3758, Y -74.6888, Z -174.0150, A 0, B 90, C 0, E1 0, E2 0, E3 0, E4 0 } C_DIS
LIN{ E6POS: X 705.6787, Y -73.7357, Z -174.0150, A 0, B 90, C 0, E1 0, E2 0, E3 0, E4 0 } C_DIS
LIN{ E6POS: X 705.8253, Y -73.2745, Z -174.0150, A 0, B 90, C 0, E1 0, E2 0, E3 0, E4 0 } C_DIS
LIN{ E6POS: X 705.8253, Y -73.2745, Z -174.0150, A 0, B 90, C 0, E1 0, E2 0, E3 0, E4 0 } C_DIS
LIN{ E6POS: X 706.1428, Y -72.3262, Z -174.0150, A 0, B 90, C 0, E1 0, E2 0, E3 0, E4 0 } C_DIS
LIN{ E6POS: X 706.2644, Y -71.9630, Z -174.0150, A 0, B 90, C 0, E1 0, E2 0, E3 0, E4 0 } C_DIS
LIN{ E6POS: X 706.2644, Y -71.9630, Z -174.0150, A 0, B 90, C 0, E1 0, E2 0, E3 0, E4 0 } C_DIS
LIN{ E6POS: X 706.5860, Y -71.0161, Z -174.0150, A 0, B 90, C 0, E1 0, E2 0, E3 0, E4 0 } C_DIS
LIN{ E6POS: X 706.6919, Y -70.7039, Z -174.0150, A 0, B 90, C 0, E1 0, E2 0, E3 0, E4 0 } C_DIS
LIN{ E6POS: X 706.6919, Y -70.7039, Z -174.0150, A 0, B 90, C 0, E1 0, E2 0, E3 0, E4 0 } C_DIS
LIN{ E6POS: X 707.0064, Y -69.7547, Z -174.0150, A 0, B 90, C 0, E1 0, E2 0, E3 0, E4 0 } C_DIS
LIN{ E6POS: X 707.1091, Y -69.4448, Z -174.0150, A 0, B 90, C 0, E1 0, E2 0, E3 0, E4 0 } C_DIS
LIN{ E6POS: X 707.1091, Y -69.4448, Z -174.0150, A 0, B 90, C 0, E1 0, E2 0, E3 0, E4 0 } C_DIS
LIN{ E6POS: X 707.4056, Y -68.4898, Z -174.0150, A 0, B 90, C 0, E1 0, E2 0, E3 0, E4 0 } C_DIS
LIN{ E6POS: X 707.5156, Y -68.1355, Z -174.0150, A 0, B 90, C 0, E1 0, E2 0, E3 0, E4 0 } C_DIS
LIN{ E6POS: X 707.5156, Y -68.1355, Z -174.0150, A 0, B 90, C 0, E1 0, E2 0, E3 0, E4 0 } C_DIS
LIN{ E6POS: X 707.7852, Y -67.1726, Z -174.0150, A 0, B 90, C 0, E1 0, E2 0, E3 0, E4 0 } C_DIS
LIN{ E6POS: X 707.9110, Y -66.7230, Z -174.0150, A 0, B 90, C 0, E1 0, E2 0, E3 0, E4 0 } C_DIS
LIN{ E6POS: X 707.9110, Y -66.7230, Z -174.0150, A 0, B 90, C 0, E1 0, E2 0, E3 0, E4 0 } C_DIS
LIN{ E6POS: X 708.1654, Y -65.7559, Z -174.0150, A 0, B 90, C 0, E1 0, E2 0, E3 0, E4 0 } C_DIS
LIN{ E6POS: X 708.2958, Y -65.2604, Z -174.0150, A 0, B 90, C 0, E1 0, E2 0, E3 0, E4 0 } C_DIS
LIN{ E6POS: X 708.2958, Y -65.2604, Z -174.0150, A 0, B 90, C 0, E1 0, E2 0, E3 0, E4 0 } C_DIS
LIN{ E6POS: X 708.5455, Y -64.2921, Z -174.0150, A 0, B 90, C 0, E1 0, E2 0, E3 0, E4 0 } C_DIS
LIN{ E6POS: X 708.6730, Y -63.7975, Z -174.0150, A 0, B 90, C 0, E1 0, E2 0, E3 0, E4 0 } C_DIS
LIN{ E6POS: X 708.6730, Y -63.7975, Z -174.0150, A 0, B 90, C 0, E1 0, E2 0, E3 0, E4 0 } C_DIS
LIN{ E6POS: X 708.9276, Y -62.8304, Z -174.0150, A 0, B 90, C 0, E1 0, E2 0, E3 0, E4 0 } C_DIS
LIN{ E6POS: X 709.0447, Y -62.3858, Z -174.0150, A 0, B 90, C 0, E1 0, E2 0, E3 0, E4 0 } C_DIS
LIN{ E6POS: X 709.0447, Y -62.3858, Z -174.0150, A 0, B 90, C 0, E1 0, E2 0, E3 0, E4 0 } C_DIS
LIN{ E6POS: X 709.3139, Y -61.4227, Z -174.0150, A 0, B 90, C 0, E1 0, E2 0, E3 0, E4 0 } C_DIS
LIN{ E6POS: X 709.4107, Y -61.0764, Z -174.0150, A 0, B 90, C 0, E1 0, E2 0, E3 0, E4 0 } C_DIS
LIN{ E6POS: X 709.4107, Y -61.0764, Z -174.0150, A 0, B 90, C 0, E1 0, E2 0, E3 0, E4 0 } C_DIS
LIN{ E6POS: X 709.6854, Y -60.1148, Z -174.0150, A 0, B 90, C 0, E1 0, E2 0, E3 0, E4 0 } C_DIS
LIN{ E6POS: X 709.7702, Y -59.8179, Z -174.0150, A 0, B 90, C 0, E1 0, E2 0, E3 0, E4 0 } C_DIS
LIN{ E6POS: X 709.7702, Y -59.8179, Z -174.0150, A 0, B 90, C 0, E1 0, E2 0, E3 0, E4 0 } C_DIS
LIN{ E6POS: X 710.0383, Y -58.8545, Z -174.0150, A 0, B 90, C 0, E1 0, E2 0, E3 0, E4 0 } C_DIS
LIN{ E6POS: X 710.1198, Y -58.5615, Z -174.0150, A 0, B 90, C 0, E1 0, E2 0, E3 0, E4 0 } C_DIS
LIN{ E6POS: X 710.1198, Y -58.5615, Z -174.0150, A 0, B 90, C 0, E1 0, E2 0, E3 0, E4 0 } C_DIS
LIN{ E6POS: X 710.3703, Y -57.5933, Z -174.0150, A 0, B 90, C 0, E1 0, E2 0, E3 0, E4 0 } C_DIS
LIN{ E6POS: X 710.4581, Y -57.2537, Z -174.0150, A 0, B 90, C 0, E1 0, E2 0, E3 0, E4 0 } C_DIS
LIN{ E6POS: X 710.4581, Y -57.2537, Z -174.0150, A 0, B 90, C 0, E1 0, E2 0, E3 0, E4 0 } C_DIS
LIN{ E6POS: X 710.6827, Y -56.2793, Z -174.0150, A 0, B 90, C 0, E1 0, E2 0, E3 0, E4 0 } C_DIS
LIN{ E6POS: X 710.7823, Y -55.8469, Z -174.0150, A 0, B 90, C 0, E1 0, E2 0, E3 0, E4 0 } C_DIS
LIN{ E6POS: X 710.7823, Y -55.8469, Z -174.0150, A 0, B 90, C 0, E1 0, E2 0, E3 0, E4 0 } C_DIS
LIN{ E6POS: X 710.9922, Y -54.8692, Z -174.0150, A 0, B 90, C 0, E1 0, E2 0, E3 0, E4 0 } C_DIS
LIN{ E6POS: X 711.0953, Y -54.3888, Z -174.0150, A 0, B 90, C 0, E1 0, E2 0, E3 0, E4 0 } C_DIS
LIN{ E6POS: X 711.0953, Y -54.3888, Z -174.0150, A 0, B 90, C 0, E1 0, E2 0, E3 0, E4 0 } C_DIS
LIN{ E6POS: X 711.3009, Y -53.4102, Z -174.0150, A 0, B 90, C 0, E1 0, E2 0, E3 0, E4 0 } C_DIS
LIN{ E6POS: X 711.4016, Y -52.9307, Z -174.0150, A 0, B 90, C 0, E1 0, E2 0, E3 0, E4 0 } C_DIS
LIN{ E6POS: X 711.4016, Y -52.9307, Z -174.0150, A 0, B 90, C 0, E1 0, E2 0, E3 0, E4 0 } C_DIS
LIN{ E6POS: X 711.6119, Y -51.9531, Z -174.0150, A 0, B 90, C 0, E1 0, E2 0, E3 0, E4 0 } C_DIS
LIN{ E6POS: X 711.7043, Y -51.5234, Z -174.0150, A 0, B 90, C 0, E1 0, E2 0, E3 0, E4 0 } C_DIS
LIN{ E6POS: X 711.7043, Y -51.5234, Z -174.0150, A 0, B 90, C 0, E1 0, E2 0, E3 0, E4 0 } C_DIS
LIN{ E6POS: X 711.9303, Y -50.5493, Z -174.0150, A 0, B 90, C 0, E1 0, E2 0, E3 0, E4 0 } C_DIS
LIN{ E6POS: X 712.0074, Y -50.2171, Z -174.0150, A 0, B 90, C 0, E1 0, E2 0, E3 0, E4 0 } C_DIS
LIN{ E6POS: X 712.0074, Y -50.2171, Z -174.0150, A 0, B 90, C 0, E1 0, E2 0, E3 0, E4 0 } C_DIS
LIN{ E6POS: X 712.2446, Y -49.2457, Z -174.0150, A 0, B 90, C 0, E1 0, E2 0, E3 0, E4 0 } C_DIS
LIN{ E6POS: X 712.3078, Y -48.9869, Z -174.0150, A 0, B 90, C 0, E1 0, E2 0, E3 0, E4 0 } C_DIS
LIN{ E6POS: X 712.3078, Y -48.9869, Z -174.0150, A 0, B 90, C 0, E1 0, E2 0, E3 0, E4 0 } C_DIS
LIN{ E6POS: X 712.5504, Y -48.0168, Z -174.0150, A 0, B 90, C 0, E1 0, E2 0, E3 0, E4 0 } C_DIS
LIN{ E6POS: X 712.6026, Y -47.8080, Z -174.0150, A 0, B 90, C 0, E1 0, E2 0, E3 0, E4 0 } C_DIS
LIN{ E6POS: X 712.6026, Y -47.8080, Z -174.0150, A 0, B 90, C 0, E1 0, E2 0, E3 0, E4 0 } C_DIS
LIN{ E6POS: X 712.8436, Y -46.8374, Z -174.0150, A 0, B 90, C 0, E1 0, E2 0, E3 0, E4 0 } C_DIS
LIN{ E6POS: X 712.8888, Y -46.6554, Z -174.0150, A 0, B 90, C 0, E1 0, E2 0, E3 0, E4 0 } C_DIS
LIN{ E6POS: X 712.8888, Y -46.6554, Z -174.0150, A 0, B 90, C 0, E1 0, E2 0, E3 0, E4 0 } C_DIS
LIN{ E6POS: X 713.1192, Y -45.6823, Z -174.0150, A 0, B 90, C 0, E1 0, E2 0, E3 0, E4 0 } C_DIS
LIN{ E6POS: X 713.1617, Y -45.5028, Z -174.0150, A 0, B 90, C 0, E1 0, E2 0, E3 0, E4 0 } C_DIS
LIN{ E6POS: X 713.1617, Y -45.5028, Z -174.0150, A 0, B 90, C 0, E1 0, E2 0, E3 0, E4 0 } C_DIS
LIN{ E6POS: X 713.3807, Y -44.5271, Z -174.0150, A 0, B 90, C 0, E1 0, E2 0, E3 0, E4 0 } C_DIS
LIN{ E6POS: X 713.4259, Y -44.3257, Z -174.0150, A 0, B 90, C 0, E1 0, E2 0, E3 0, E4 0 } C_DIS
LIN{ E6POS: X 713.4259, Y -44.3257, Z -174.0150, A 0, B 90, C 0, E1 0, E2 0, E3 0, E4 0 } C_DIS
LIN{ E6POS: X 713.6296, Y -43.3467, Z -174.0150, A 0, B 90, C 0, E1 0, E2 0, E3 0, E4 0 } C_DIS
LIN{ E6POS: X 713.6809, Y -43.1000, Z -174.0150, A 0, B 90, C 0, E1 0, E2 0, E3 0, E4 0 } C_DIS
LIN{ E6POS: X 713.6809, Y -43.1000, Z -174.0150, A 0, B 90, C 0, E1 0, E2 0, E3 0, E4 0 } C_DIS
LIN{ E6POS: X 713.8696, Y -42.1179, Z -174.0150, A 0, B 90, C 0, E1 0, E2 0, E3 0, E4 0 } C_DIS
LIN{ E6POS: X 713.9309, Y -41.7988, Z -174.0150, A 0, B 90, C 0, E1 0, E2 0, E3 0, E4 0 } C_DIS
LIN{ E6POS: X 713.9309, Y -41.7988, Z -174.0150, A 0, B 90, C 0, E1 0, E2 0, E3 0, E4 0 } C_DIS
LIN{ E6POS: X 714.1034, Y -40.8138, Z -174.0150, A 0, B 90, C 0, E1 0, E2 0, E3 0, E4 0 } C_DIS
LIN{ E6POS: X 714.1762, Y -40.3985, Z -174.0150, A 0, B 90, C 0, E1 0, E2 0, E3 0, E4 0 } C_DIS
LIN{ E6POS: X 714.1762, Y -40.3985, Z -174.0150, A 0, B 90, C 0, E1 0, E2 0, E3 0, E4 0 } C_DIS
LIN{ E6POS: X 714.3397, Y -39.4120, Z -174.0150, A 0, B 90, C 0, E1 0, E2 0, E3 0, E4 0 } C_DIS
LIN{ E6POS: X 714.4166, Y -38.9478, Z -174.0150, A 0, B 90, C 0, E1 0, E2 0, E3 0, E4 0 } C_DIS
LIN{ E6POS: X 714.4166, Y -38.9478, Z -174.0150, A 0, B 90, C 0, E1 0, E2 0, E3 0, E4 0 } C_DIS
LIN{ E6POS: X 714.5768, Y -37.9608, Z -174.0150, A 0, B 90, C 0, E1 0, E2 0, E3 0, E4 0 } C_DIS
LIN{ E6POS: X 714.6518, Y -37.4987, Z -174.0150, A 0, B 90, C 0, E1 0, E2 0, E3 0, E4 0 } C_DIS
LIN{ E6POS: X 714.6518, Y -37.4987, Z -174.0150, A 0, B 90, C 0, E1 0, E2 0, E3 0, E4 0 } C_DIS
LIN{ E6POS: X 714.8140, Y -36.5119, Z -174.0150, A 0, B 90, C 0, E1 0, E2 0, E3 0, E4 0 } C_DIS
LIN{ E6POS: X 714.8817, Y -36.0998, Z -174.0150, A 0, B 90, C 0, E1 0, E2 0, E3 0, E4 0 } C_DIS
LIN{ E6POS: X 714.8817, Y -36.0998, Z -174.0150, A 0, B 90, C 0, E1 0, E2 0, E3 0, E4 0 } C_DIS
LIN{ E6POS: X 715.0523, Y -35.1144, Z -174.0150, A 0, B 90, C 0, E1 0, E2 0, E3 0, E4 0 } C_DIS
LIN{ E6POS: X 715.1065, Y -34.8011, Z -174.0150, A 0, B 90, C 0, E1 0, E2 0, E3 0, E4 0 } C_DIS
LIN{ E6POS: X 715.1065, Y -34.8011, Z -174.0150, A 0, B 90, C 0, E1 0, E2 0, E3 0, E4 0 } C_DIS
LIN{ E6POS: X 715.2788, Y -33.8161, Z -174.0150, A 0, B 90, C 0, E1 0, E2 0, E3 0, E4 0 } C_DIS
LIN{ E6POS: X 715.3248, Y -33.5535, Z -174.0150, A 0, B 90, C 0, E1 0, E2 0, E3 0, E4 0 } C_DIS
LIN{ E6POS: X 715.3248, Y -33.5535, Z -174.0150, A 0, B 90, C 0, E1 0, E2 0, E3 0, E4 0 } C_DIS
LIN{ E6POS: X 715.4919, Y -32.5676, Z -174.0150, A 0, B 90, C 0, E1 0, E2 0, E3 0, E4 0 } C_DIS
LIN{ E6POS: X 715.5360, Y -32.3078, Z -174.0150, A 0, B 90, C 0, E1 0, E2 0, E3 0, E4 0 } C_DIS
LIN{ E6POS: X 715.5360, Y -32.3078, Z -174.0150, A 0, B 90, C 0, E1 0, E2 0, E3 0, E4 0 } C_DIS
LIN{ E6POS: X 715.6923, Y -31.3201, Z -174.0150, A 0, B 90, C 0, E1 0, E2 0, E3 0, E4 0 } C_DIS
LIN{ E6POS: X 715.7409, Y -31.0133, Z -174.0150, A 0, B 90, C 0, E1 0, E2 0, E3 0, E4 0 } C_DIS
LIN{ E6POS: X 715.7409, Y -31.0133, Z -174.0150, A 0, B 90, C 0, E1 0, E2 0, E3 0, E4 0 } C_DIS
LIN{ E6POS: X 715.8816, Y -30.0233, Z -174.0150, A 0, B 90, C 0, E1 0, E2 0, E3 0, E4 0 } C_DIS
LIN{ E6POS: X 715.9386, Y -29.6220, Z -174.0150, A 0, B 90, C 0, E1 0, E2 0, E3 0, E4 0 } C_DIS
LIN{ E6POS: X 715.9386, Y -29.6220, Z -174.0150, A 0, B 90, C 0, E1 0, E2 0, E3 0, E4 0 } C_DIS
LIN{ E6POS: X 716.0705, Y -28.6308, Z -174.0150, A 0, B 90, C 0, E1 0, E2 0, E3 0, E4 0 } C_DIS
LIN{ E6POS: X 716.1304, Y -28.1811, Z -174.0150, A 0, B 90, C 0, E1 0, E2 0, E3 0, E4 0 } C_DIS
LIN{ E6POS: X 716.1304, Y -28.1811, Z -174.0150, A 0, B 90, C 0, E1 0, E2 0, E3 0, E4 0 } C_DIS
LIN{ E6POS: X 716.2595, Y -27.1894, Z -174.0150, A 0, B 90, C 0, E1 0, E2 0, E3 0, E4 0 } C_DIS
LIN{ E6POS: X 716.3179, Y -26.7419, Z -174.0150, A 0, B 90, C 0, E1 0, E2 0, E3 0, E4 0 } C_DIS
LIN{ E6POS: X 716.3179, Y -26.7419, Z -174.0150, A 0, B 90, C 0, E1 0, E2 0, E3 0, E4 0 } C_DIS
LIN{ E6POS: X 716.4506, Y -25.7507, Z -174.0150, A 0, B 90, C 0, E1 0, E2 0, E3 0, E4 0 } C_DIS
LIN{ E6POS: X 716.5042, Y -25.3511, Z -174.0150, A 0, B 90, C 0, E1 0, E2 0, E3 0, E4 0 } C_DIS
LIN{ E6POS: X 716.5042, Y -25.3511, Z -174.0150, A 0, B 90, C 0, E1 0, E2 0, E3 0, E4 0 } C_DIS
LIN{ E6POS: X 716.6455, Y -24.3612, Z -174.0150, A 0, B 90, C 0, E1 0, E2 0, E3 0, E4 0 } C_DIS
LIN{ E6POS: X 716.6885, Y -24.0596, Z -174.0150, A 0, B 90, C 0, E1 0, E2 0, E3 0, E4 0 } C_DIS
LIN{ E6POS: X 716.6885, Y -24.0596, Z -174.0150, A 0, B 90, C 0, E1 0, E2 0, E3 0, E4 0 } C_DIS
LIN{ E6POS: X 716.8346, Y -23.0703, Z -174.0150, A 0, B 90, C 0, E1 0, E2 0, E3 0, E4 0 } C_DIS
LIN{ E6POS: X 716.8686, Y -22.8395, Z -174.0150, A 0, B 90, C 0, E1 0, E2 0, E3 0, E4 0 } C_DIS
LIN{ E6POS: X 716.8686, Y -22.8395, Z -174.0150, A 0, B 90, C 0, E1 0, E2 0, E3 0, E4 0 } C_DIS
LIN{ E6POS: X 717.0123, Y -21.8499, Z -174.0150, A 0, B 90, C 0, E1 0, E2 0, E3 0, E4 0 } C_DIS
LIN{ E6POS: X 717.0394, Y -21.6632, Z -174.0150, A 0, B 90, C 0, E1 0, E2 0, E3 0, E4 0 } C_DIS
LIN{ E6POS: X 717.0394, Y -21.6632, Z -174.0150, A 0, B 90, C 0, E1 0, E2 0, E3 0, E4 0 } C_DIS
LIN{ E6POS: X 717.1738, Y -20.6723, Z -174.0150, A 0, B 90, C 0, E1 0, E2 0, E3 0, E4 0 } C_DIS
LIN{ E6POS: X 717.1969, Y -20.5016, Z -174.0150, A 0, B 90, C 0, E1 0, E2 0, E3 0, E4 0 } C_DIS
LIN{ E6POS: X 717.1969, Y -20.5016, Z -174.0150, A 0, B 90, C 0, E1 0, E2 0, E3 0, E4 0 } C_DIS
LIN{ E6POS: X 717.3160, Y -19.5087, Z -174.0150, A 0, B 90, C 0, E1 0, E2 0, E3 0, E4 0 } C_DIS
LIN{ E6POS: X 717.3376, Y -19.3284, Z -174.0150, A 0, B 90, C 0, E1 0, E2 0, E3 0, E4 0 } C_DIS
LIN{ E6POS: X 717.3376, Y -19.3284, Z -174.0150, A 0, B 90, C 0, E1 0, E2 0, E3 0, E4 0 } C_DIS
LIN{ E6POS: X 717.4445, Y -18.3341, Z -174.0150, A 0, B 90, C 0, E1 0, E2 0, E3 0, E4 0 } C_DIS
LIN{ E6POS: X 717.4648, Y -18.1457, Z -174.0150, A 0, B 90, C 0, E1 0, E2 0, E3 0, E4 0 } C_DIS
LIN{ E6POS: X 717.4648, Y -18.1457, Z -174.0150, A 0, B 90, C 0, E1 0, E2 0, E3 0, E4 0 } C_DIS
LIN{ E6POS: X 717.5638, Y -17.1507, Z -174.0150, A 0, B 90, C 0, E1 0, E2 0, E3 0, E4 0 } C_DIS
LIN{ E6POS: X 717.5831, Y -16.9572, Z -174.0150, A 0, B 90, C 0, E1 0, E2 0, E3 0, E4 0 } C_DIS
LIN{ E6POS: X 717.5831, Y -16.9572, Z -174.0150, A 0, B 90, C 0, E1 0, E2 0, E3 0, E4 0 } C_DIS
LIN{ E6POS: X 717.6859, Y -15.9625, Z -174.0150, A 0, B 90, C 0, E1 0, E2 0, E3 0, E4 0 } C_DIS
LIN{ E6POS: X 717.7887, Y -14.9678, Z -174.0150, A 0, B 90, C 0, E1 0, E2 0, E3 0, E4 0 } C_DIS
LIN{ E6POS: X 717.8058, Y -14.8024, Z -174.0150, A 0, B 90, C 0, E1 0, E2 0, E3 0, E4 0 } C_DIS
LIN{ E6POS: X 717.8058, Y -14.8024, Z -174.0150, A 0, B 90, C 0, E1 0, E2 0, E3 0, E4 0 } C_DIS
LIN{ E6POS: X 717.9316, Y -13.8104, Z -174.0150, A 0, B 90, C 0, E1 0, E2 0, E3 0, E4 0 } C_DIS
LIN{ E6POS: X 718.0574, Y -12.8183, Z -174.0150, A 0, B 90, C 0, E1 0, E2 0, E3 0, E4 0 } C_DIS
LIN{ E6POS: X 718.1499, Y -12.0880, Z -174.0150, A 0, B 90, C 0, E1 0, E2 0, E3 0, E4 0 } C_DIS
LIN{ E6POS: X 718.1499, Y -12.0880, Z -174.0150, A 0, B 90, C 0, E1 0, E2 0, E3 0, E4 0 } C_DIS
LIN{ E6POS: X 718.2726, Y -11.0955, Z -174.0150, A 0, B 90, C 0, E1 0, E2 0, E3 0, E4 0 } C_DIS
LIN{ E6POS: X 718.2928, Y -10.9321, Z -174.0150, A 0, B 90, C 0, E1 0, E2 0, E3 0, E4 0 } C_DIS
LIN{ E6POS: X 718.2928, Y -10.9321, Z -174.0150, A 0, B 90, C 0, E1 0, E2 0, E3 0, E4 0 } C_DIS
LIN{ E6POS: X 718.4047, Y -9.9384, Z -174.0150, A 0, B 90, C 0, E1 0, E2 0, E3 0, E4 0 } C_DIS
LIN{ E6POS: X 718.4365, Y -9.6559, Z -174.0150, A 0, B 90, C 0, E1 0, E2 0, E3 0, E4 0 } C_DIS
LIN{ E6POS: X 718.4365, Y -9.6559, Z -174.0150, A 0, B 90, C 0, E1 0, E2 0, E3 0, E4 0 } C_DIS
LIN{ E6POS: X 718.5335, Y -8.6606, Z -174.0150, A 0, B 90, C 0, E1 0, E2 0, E3 0, E4 0 } C_DIS
LIN{ E6POS: X 718.5698, Y -8.2880, Z -174.0150, A 0, B 90, C 0, E1 0, E2 0, E3 0, E4 0 } C_DIS
LIN{ E6POS: X 718.5698, Y -8.2880, Z -174.0150, A 0, B 90, C 0, E1 0, E2 0, E3 0, E4 0 } C_DIS
LIN{ E6POS: X 718.6589, Y -7.2920, Z -174.0150, A 0, B 90, C 0, E1 0, E2 0, E3 0, E4 0 } C_DIS
LIN{ E6POS: X 718.6964, Y -6.8734, Z -174.0150, A 0, B 90, C 0, E1 0, E2 0, E3 0, E4 0 } C_DIS
LIN{ E6POS: X 718.6964, Y -6.8734, Z -174.0150, A 0, B 90, C 0, E1 0, E2 0, E3 0, E4 0 } C_DIS
LIN{ E6POS: X 718.7841, Y -5.8773, Z -174.0150, A 0, B 90, C 0, E1 0, E2 0, E3 0, E4 0 } C_DIS
LIN{ E6POS: X 718.8209, Y -5.4592, Z -174.0150, A 0, B 90, C 0, E1 0, E2 0, E3 0, E4 0 } C_DIS
LIN{ E6POS: X 718.8209, Y -5.4592, Z -174.0150, A 0, B 90, C 0, E1 0, E2 0, E3 0, E4 0 } C_DIS
LIN{ E6POS: X 718.9136, Y -4.4635, Z -174.0150, A 0, B 90, C 0, E1 0, E2 0, E3 0, E4 0 } C_DIS
LIN{ E6POS: X 718.9480, Y -4.0936, Z -174.0150, A 0, B 90, C 0, E1 0, E2 0, E3 0, E4 0 } C_DIS
LIN{ E6POS: X 718.9480, Y -4.0936, Z -174.0150, A 0, B 90, C 0, E1 0, E2 0, E3 0, E4 0 } C_DIS
LIN{ E6POS: X 719.0528, Y -3.0991, Z -174.0150, A 0, B 90, C 0, E1 0, E2 0, E3 0, E4 0 } C_DIS
LIN{ E6POS: X 719.0819, Y -2.8226, Z -174.0150, A 0, B 90, C 0, E1 0, E2 0, E3 0, E4 0 } C_DIS
LIN{ E6POS: X 719.0819, Y -2.8226, Z -174.0150, A 0, B 90, C 0, E1 0, E2 0, E3 0, E4 0 } C_DIS
LIN{ E6POS: X 719.1922, Y -1.8287, Z -174.0150, A 0, B 90, C 0, E1 0, E2 0, E3 0, E4 0 } C_DIS
LIN{ E6POS: X 719.2177, Y -1.5990, Z -174.0150, A 0, B 90, C 0, E1 0, E2 0, E3 0, E4 0 } C_DIS
LIN{ E6POS: X 719.2177, Y -1.5990, Z -174.0150, A 0, B 90, C 0, E1 0, E2 0, E3 0, E4 0 } C_DIS
LIN{ E6POS: X 719.3269, Y -0.6050, Z -174.0150, A 0, B 90, C 0, E1 0, E2 0, E3 0, E4 0 } C_DIS
LIN{ E6POS: X 719.3519, Y -0.3780, Z -174.0150, A 0, B 90, C 0, E1 0, E2 0, E3 0, E4 0 } C_DIS
LIN{ E6POS: X 719.3519, Y -0.3780, Z -174.0150, A 0, B 90, C 0, E1 0, E2 0, E3 0, E4 0 } C_DIS
LIN{ E6POS: X 719.4514, Y 0.6170, Z -174.0150, A 0, B 90, C 0, E1 0, E2 0, E3 0, E4 0 } C_DIS
LIN{ E6POS: X 719.4783, Y 0.8859, Z -174.0150, A 0, B 90, C 0, E1 0, E2 0, E3 0, E4 0 } C_DIS
LIN{ E6POS: X 719.4783, Y 0.8859, Z -174.0150, A 0, B 90, C 0, E1 0, E2 0, E3 0, E4 0 } C_DIS
LIN{ E6POS: X 719.5633, Y 1.8823, Z -174.0150, A 0, B 90, C 0, E1 0, E2 0, E3 0, E4 0 } C_DIS
LIN{ E6POS: X 719.5938, Y 2.2395, Z -174.0150, A 0, B 90, C 0, E1 0, E2 0, E3 0, E4 0 } C_DIS
LIN{ E6POS: X 719.5938, Y 2.2395, Z -174.0150, A 0, B 90, C 0, E1 0, E2 0, E3 0, E4 0 } C_DIS
LIN{ E6POS: X 719.6723, Y 3.2365, Z -174.0150, A 0, B 90, C 0, E1 0, E2 0, E3 0, E4 0 } C_DIS
LIN{ E6POS: X 719.7038, Y 3.6375, Z -174.0150, A 0, B 90, C 0, E1 0, E2 0, E3 0, E4 0 } C_DIS
LIN{ E6POS: X 719.7038, Y 3.6375, Z -174.0150, A 0, B 90, C 0, E1 0, E2 0, E3 0, E4 0 } C_DIS
LIN{ E6POS: X 719.7815, Y 4.6345, Z -174.0150, A 0, B 90, C 0, E1 0, E2 0, E3 0, E4 0 } C_DIS
LIN{ E6POS: X 719.8127, Y 5.0348, Z -174.0150, A 0, B 90, C 0, E1 0, E2 0, E3 0, E4 0 } C_DIS
LIN{ E6POS: X 719.8127, Y 5.0348, Z -174.0150, A 0, B 90, C 0, E1 0, E2 0, E3 0, E4 0 } C_DIS
LIN{ E6POS: X 719.8960, Y 6.0314, Z -174.0150, A 0, B 90, C 0, E1 0, E2 0, E3 0, E4 0 } C_DIS
LIN{ E6POS: X 719.9255, Y 6.3852, Z -174.0150, A 0, B 90, C 0, E1 0, E2 0, E3 0, E4 0 } C_DIS
LIN{ E6POS: X 719.9255, Y 6.3852, Z -174.0150, A 0, B 90, C 0, E1 0, E2 0, E3 0, E4 0 } C_DIS
LIN{ E6POS: X 720.0222, Y 7.3805, Z -174.0150, A 0, B 90, C 0, E1 0, E2 0, E3 0, E4 0 } C_DIS
LIN{ E6POS: X 720.0478, Y 7.6442, Z -174.0150, A 0, B 90, C 0, E1 0, E2 0, E3 0, E4 0 } C_DIS
LIN{ E6POS: X 720.0478, Y 7.6442, Z -174.0150, A 0, B 90, C 0, E1 0, E2 0, E3 0, E4 0 } C_DIS
LIN{ E6POS: X 720.1514, Y 8.6388, Z -174.0150, A 0, B 90, C 0, E1 0, E2 0, E3 0, E4 0 } C_DIS
LIN{ E6POS: X 720.1741, Y 8.8562, Z -174.0150, A 0, B 90, C 0, E1 0, E2 0, E3 0, E4 0 } C_DIS
LIN{ E6POS: X 720.1741, Y 8.8562, Z -174.0150, A 0, B 90, C 0, E1 0, E2 0, E3 0, E4 0 } C_DIS
LIN{ E6POS: X 720.2773, Y 9.8508, Z -174.0150, A 0, B 90, C 0, E1 0, E2 0, E3 0, E4 0 } C_DIS
LIN{ E6POS: X 720.2995, Y 10.0653, Z -174.0150, A 0, B 90, C 0, E1 0, E2 0, E3 0, E4 0 } C_DIS
LIN{ E6POS: X 720.2995, Y 10.0653, Z -174.0150, A 0, B 90, C 0, E1 0, E2 0, E3 0, E4 0 } C_DIS
LIN{ E6POS: X 720.3945, Y 11.0608, Z -174.0150, A 0, B 90, C 0, E1 0, E2 0, E3 0, E4 0 } C_DIS
LIN{ E6POS: X 720.4190, Y 11.3169, Z -174.0150, A 0, B 90, C 0, E1 0, E2 0, E3 0, E4 0 } C_DIS
LIN{ E6POS: X 720.4190, Y 11.3169, Z -174.0150, A 0, B 90, C 0, E1 0, E2 0, E3 0, E4 0 } C_DIS
LIN{ E6POS: X 720.5005, Y 12.3136, Z -174.0150, A 0, B 90, C 0, E1 0, E2 0, E3 0, E4 0 } C_DIS
LIN{ E6POS: X 720.5283, Y 12.6538, Z -174.0150, A 0, B 90, C 0, E1 0, E2 0, E3 0, E4 0 } C_DIS
LIN{ E6POS: X 720.5283, Y 12.6538, Z -174.0150, A 0, B 90, C 0, E1 0, E2 0, E3 0, E4 0 } C_DIS
LIN{ E6POS: X 720.6030, Y 13.6510, Z -174.0150, A 0, B 90, C 0, E1 0, E2 0, E3 0, E4 0 } C_DIS
LIN{ E6POS: X 720.6317, Y 14.0331, Z -174.0150, A 0, B 90, C 0, E1 0, E2 0, E3 0, E4 0 } C_DIS
LIN{ E6POS: X 720.6317, Y 14.0331, Z -174.0150, A 0, B 90, C 0, E1 0, E2 0, E3 0, E4 0 } C_DIS
LIN{ E6POS: X 720.7064, Y 15.0303, Z -174.0150, A 0, B 90, C 0, E1 0, E2 0, E3 0, E4 0 } C_DIS
LIN{ E6POS: X 720.7350, Y 15.4124, Z -174.0150, A 0, B 90, C 0, E1 0, E2 0, E3 0, E4 0 } C_DIS
LIN{ E6POS: X 720.7350, Y 15.4124, Z -174.0150, A 0, B 90, C 0, E1 0, E2 0, E3 0, E4 0 } C_DIS
LIN{ E6POS: X 720.8161, Y 16.4091, Z -174.0150, A 0, B 90, C 0, E1 0, E2 0, E3 0, E4 0 } C_DIS
LIN{ E6POS: X 720.8436, Y 16.7463, Z -174.0150, A 0, B 90, C 0, E1 0, E2 0, E3 0, E4 0 } C_DIS
LIN{ E6POS: X 720.8436, Y 16.7463, Z -174.0150, A 0, B 90, C 0, E1 0, E2 0, E3 0, E4 0 } C_DIS
LIN{ E6POS: X 720.9399, Y 17.7417, Z -174.0150, A 0, B 90, C 0, E1 0, E2 0, E3 0, E4 0 } C_DIS
LIN{ E6POS: X 720.9639, Y 17.9904, Z -174.0150, A 0, B 90, C 0, E1 0, E2 0, E3 0, E4 0 } C_DIS
LIN{ E6POS: X 720.9639, Y 17.9904, Z -174.0150, A 0, B 90, C 0, E1 0, E2 0, E3 0, E4 0 } C_DIS
LIN{ E6POS: X 721.0683, Y 18.9849, Z -174.0150, A 0, B 90, C 0, E1 0, E2 0, E3 0, E4 0 } C_DIS
LIN{ E6POS: X 721.0898, Y 19.1900, Z -174.0150, A 0, B 90, C 0, E1 0, E2 0, E3 0, E4 0 } C_DIS
LIN{ E6POS: X 721.0898, Y 19.1900, Z -174.0150, A 0, B 90, C 0, E1 0, E2 0, E3 0, E4 0 } C_DIS
LIN{ E6POS: X 721.1944, Y 20.1845, Z -174.0150, A 0, B 90, C 0, E1 0, E2 0, E3 0, E4 0 } C_DIS
LIN{ E6POS: X 721.2156, Y 20.3856, Z -174.0150, A 0, B 90, C 0, E1 0, E2 0, E3 0, E4 0 } C_DIS
LIN{ E6POS: X 721.2156, Y 20.3856, Z -174.0150, A 0, B 90, C 0, E1 0, E2 0, E3 0, E4 0 } C_DIS
LIN{ E6POS: X 721.3138, Y 21.3807, Z -174.0150, A 0, B 90, C 0, E1 0, E2 0, E3 0, E4 0 } C_DIS
LIN{ E6POS: X 721.3376, Y 21.6218, Z -174.0150, A 0, B 90, C 0, E1 0, E2 0, E3 0, E4 0 } C_DIS
LIN{ E6POS: X 721.3376, Y 21.6218, Z -174.0150, A 0, B 90, C 0, E1 0, E2 0, E3 0, E4 0 } C_DIS
LIN{ E6POS: X 721.4217, Y 22.6182, Z -174.0150, A 0, B 90, C 0, E1 0, E2 0, E3 0, E4 0 } C_DIS
LIN{ E6POS: X 721.4489, Y 22.9404, Z -174.0150, A 0, B 90, C 0, E1 0, E2 0, E3 0, E4 0 } C_DIS
LIN{ E6POS: X 721.4489, Y 22.9404, Z -174.0150, A 0, B 90, C 0, E1 0, E2 0, E3 0, E4 0 } C_DIS
LIN{ E6POS: X 721.5279, Y 23.9372, Z -174.0150, A 0, B 90, C 0, E1 0, E2 0, E3 0, E4 0 } C_DIS
LIN{ E6POS: X 721.5567, Y 24.3006, Z -174.0150, A 0, B 90, C 0, E1 0, E2 0, E3 0, E4 0 } C_DIS
LIN{ E6POS: X 721.5567, Y 24.3006, Z -174.0150, A 0, B 90, C 0, E1 0, E2 0, E3 0, E4 0 } C_DIS
LIN{ E6POS: X 721.6368, Y 25.2974, Z -174.0150, A 0, B 90, C 0, E1 0, E2 0, E3 0, E4 0 } C_DIS
LIN{ E6POS: X 721.6658, Y 25.6583, Z -174.0150, A 0, B 90, C 0, E1 0, E2 0, E3 0, E4 0 } C_DIS
LIN{ E6POS: X 721.6658, Y 25.6583, Z -174.0150, A 0, B 90, C 0, E1 0, E2 0, E3 0, E4 0 } C_DIS
LIN{ E6POS: X 721.7529, Y 26.6545, Z -174.0150, A 0, B 90, C 0, E1 0, E2 0, E3 0, E4 0 } C_DIS
LIN{ E6POS: X 721.7807, Y 26.9727, Z -174.0150, A 0, B 90, C 0, E1 0, E2 0, E3 0, E4 0 } C_DIS
LIN{ E6POS: X 721.7807, Y 26.9727, Z -174.0150, A 0, B 90, C 0, E1 0, E2 0, E3 0, E4 0 } C_DIS
LIN{ E6POS: X 721.8834, Y 27.9674, Z -174.0150, A 0, B 90, C 0, E1 0, E2 0, E3 0, E4 0 } C_DIS
LIN{ E6POS: X 721.9076, Y 28.2021, Z -174.0150, A 0, B 90, C 0, E1 0, E2 0, E3 0, E4 0 } C_DIS
LIN{ E6POS: X 721.9076, Y 28.2021, Z -174.0150, A 0, B 90, C 0, E1 0, E2 0, E3 0, E4 0 } C_DIS
LIN{ E6POS: X 722.0202, Y 29.1958, Z -174.0150, A 0, B 90, C 0, E1 0, E2 0, E3 0, E4 0 } C_DIS
LIN{ E6POS: X 722.0418, Y 29.3867, Z -174.0150, A 0, B 90, C 0, E1 0, E2 0, E3 0, E4 0 } C_DIS
LIN{ E6POS: X 722.0418, Y 29.3867, Z -174.0150, A 0, B 90, C 0, E1 0, E2 0, E3 0, E4 0 } C_DIS
LIN{ E6POS: X 722.1564, Y 30.3801, Z -174.0150, A 0, B 90, C 0, E1 0, E2 0, E3 0, E4 0 } C_DIS
LIN{ E6POS: X 722.1780, Y 30.5676, Z -174.0150, A 0, B 90, C 0, E1 0, E2 0, E3 0, E4 0 } C_DIS
LIN{ E6POS: X 722.1780, Y 30.5676, Z -174.0150, A 0, B 90, C 0, E1 0, E2 0, E3 0, E4 0 } C_DIS
LIN{ E6POS: X 722.2862, Y 31.5617, Z -174.0150, A 0, B 90, C 0, E1 0, E2 0, E3 0, E4 0 } C_DIS
LIN{ E6POS: X 722.3108, Y 31.7869, Z -174.0150, A 0, B 90, C 0, E1 0, E2 0, E3 0, E4 0 } C_DIS
LIN{ E6POS: X 722.3108, Y 31.7869, Z -174.0150, A 0, B 90, C 0, E1 0, E2 0, E3 0, E4 0 } C_DIS
LIN{ E6POS: X 722.4066, Y 32.7823, Z -174.0150, A 0, B 90, C 0, E1 0, E2 0, E3 0, E4 0 } C_DIS
LIN{ E6POS: X 722.4357, Y 33.0856, Z -174.0150, A 0, B 90, C 0, E1 0, E2 0, E3 0, E4 0 } C_DIS
LIN{ E6POS: X 722.4357, Y 33.0856, Z -174.0150, A 0, B 90, C 0, E1 0, E2 0, E3 0, E4 0 } C_DIS
LIN{ E6POS: X 722.5265, Y 34.0815, Z -174.0150, A 0, B 90, C 0, E1 0, E2 0, E3 0, E4 0 } C_DIS
LIN{ E6POS: X 722.5577, Y 34.4237, Z -174.0150, A 0, B 90, C 0, E1 0, E2 0, E3 0, E4 0 } C_DIS
LIN{ E6POS: X 722.5577, Y 34.4237, Z -174.0150, A 0, B 90, C 0, E1 0, E2 0, E3 0, E4 0 } C_DIS
LIN{ E6POS: X 722.6502, Y 35.4194, Z -174.0150, A 0, B 90, C 0, E1 0, E2 0, E3 0, E4 0 } C_DIS
LIN{ E6POS: X 722.6817, Y 35.7591, Z -174.0150, A 0, B 90, C 0, E1 0, E2 0, E3 0, E4 0 } C_DIS
LIN{ E6POS: X 722.6817, Y 35.7591, Z -174.0150, A 0, B 90, C 0, E1 0, E2 0, E3 0, E4 0 } C_DIS
LIN{ E6POS: X 722.7833, Y 36.7539, Z -174.0150, A 0, B 90, C 0, E1 0, E2 0, E3 0, E4 0 } C_DIS
LIN{ E6POS: X 722.8138, Y 37.0525, Z -174.0150, A 0, B 90, C 0, E1 0, E2 0, E3 0, E4 0 } C_DIS
LIN{ E6POS: X 722.8138, Y 37.0525, Z -174.0150, A 0, B 90, C 0, E1 0, E2 0, E3 0, E4 0 } C_DIS
LIN{ E6POS: X 722.9317, Y 38.0455, Z -174.0150, A 0, B 90, C 0, E1 0, E2 0, E3 0, E4 0 } C_DIS
LIN{ E6POS: X 722.9576, Y 38.2632, Z -174.0150, A 0, B 90, C 0, E1 0, E2 0, E3 0, E4 0 } C_DIS
LIN{ E6POS: X 722.9576, Y 38.2632, Z -174.0150, A 0, B 90, C 0, E1 0, E2 0, E3 0, E4 0 } C_DIS
LIN{ E6POS: X 723.0856, Y 39.2549, Z -174.0150, A 0, B 90, C 0, E1 0, E2 0, E3 0, E4 0 } C_DIS
LIN{ E6POS: X 723.1085, Y 39.4321, Z -174.0150, A 0, B 90, C 0, E1 0, E2 0, E3 0, E4 0 } C_DIS
LIN{ E6POS: X 723.1085, Y 39.4321, Z -174.0150, A 0, B 90, C 0, E1 0, E2 0, E3 0, E4 0 } C_DIS
LIN{ E6POS: X 723.2408, Y 40.4233, Z -174.0150, A 0, B 90, C 0, E1 0, E2 0, E3 0, E4 0 } C_DIS
LIN{ E6POS: X 723.2639, Y 40.5965, Z -174.0150, A 0, B 90, C 0, E1 0, E2 0, E3 0, E4 0 } C_DIS
LIN{ E6POS: X 723.2639, Y 40.5965, Z -174.0150, A 0, B 90, C 0, E1 0, E2 0, E3 0, E4 0 } C_DIS
LIN{ E6POS: X 723.3907, Y 41.5885, Z -174.0150, A 0, B 90, C 0, E1 0, E2 0, E3 0, E4 0 } C_DIS
LIN{ E6POS: X 723.4173, Y 41.7969, Z -174.0150, A 0, B 90, C 0, E1 0, E2 0, E3 0, E4 0 } C_DIS
LIN{ E6POS: X 723.4173, Y 41.7969, Z -174.0150, A 0, B 90, C 0, E1 0, E2 0, E3 0, E4 0 } C_DIS
LIN{ E6POS: X 723.5329, Y 42.7902, Z -174.0150, A 0, B 90, C 0, E1 0, E2 0, E3 0, E4 0 } C_DIS
LIN{ E6POS: X 723.5659, Y 43.0737, Z -174.0150, A 0, B 90, C 0, E1 0, E2 0, E3 0, E4 0 } C_DIS
LIN{ E6POS: X 723.5659, Y 43.0737, Z -174.0150, A 0, B 90, C 0, E1 0, E2 0, E3 0, E4 0 } C_DIS
LIN{ E6POS: X 723.6769, Y 44.0675, Z -174.0150, A 0, B 90, C 0, E1 0, E2 0, E3 0, E4 0 } C_DIS
LIN{ E6POS: X 723.7126, Y 44.3874, Z -174.0150, A 0, B 90, C 0, E1 0, E2 0, E3 0, E4 0 } C_DIS
LIN{ E6POS: X 723.7126, Y 44.3874, Z -174.0150, A 0, B 90, C 0, E1 0, E2 0, E3 0, E4 0 } C_DIS
LIN{ E6POS: X 723.8247, Y 45.3811, Z -174.0150, A 0, B 90, C 0, E1 0, E2 0, E3 0, E4 0 } C_DIS
LIN{ E6POS: X 723.8606, Y 45.6987, Z -174.0150, A 0, B 90, C 0, E1 0, E2 0, E3 0, E4 0 } C_DIS
LIN{ E6POS: X 723.8606, Y 45.6987, Z -174.0150, A 0, B 90, C 0, E1 0, E2 0, E3 0, E4 0 } C_DIS
LIN{ E6POS: X 723.9814, Y 46.6913, Z -174.0150, A 0, B 90, C 0, E1 0, E2 0, E3 0, E4 0 } C_DIS
LIN{ E6POS: X 724.0153, Y 46.9704, Z -174.0150, A 0, B 90, C 0, E1 0, E2 0, E3 0, E4 0 } C_DIS
LIN{ E6POS: X 724.0153, Y 46.9704, Z -174.0150, A 0, B 90, C 0, E1 0, E2 0, E3 0, E4 0 } C_DIS
LIN{ E6POS: X 724.1507, Y 47.9612, Z -174.0150, A 0, B 90, C 0, E1 0, E2 0, E3 0, E4 0 } C_DIS
LIN{ E6POS: X 724.1784, Y 48.1646, Z -174.0150, A 0, B 90, C 0, E1 0, E2 0, E3 0, E4 0 } C_DIS
LIN{ E6POS: X 724.1784, Y 48.1646, Z -174.0150, A 0, B 90, C 0, E1 0, E2 0, E3 0, E4 0 } C_DIS
LIN{ E6POS: X 724.3277, Y 49.1534, Z -174.0150, A 0, B 90, C 0, E1 0, E2 0, E3 0, E4 0 } C_DIS
LIN{ E6POS: X 724.3497, Y 49.2991, Z -174.0150, A 0, B 90, C 0, E1 0, E2 0, E3 0, E4 0 } C_DIS
LIN{ E6POS: X 724.3497, Y 49.2991, Z -174.0150, A 0, B 90, C 0, E1 0, E2 0, E3 0, E4 0 } C_DIS
LIN{ E6POS: X 724.5078, Y 50.2865, Z -174.0150, A 0, B 90, C 0, E1 0, E2 0, E3 0, E4 0 } C_DIS
LIN{ E6POS: X 724.5252, Y 50.3949, Z -174.0150, A 0, B 90, C 0, E1 0, E2 0, E3 0, E4 0 } C_DIS
LIN{ E6POS: X 724.5252, Y 50.3949, Z -174.0150, A 0, B 90, C 0, E1 0, E2 0, E3 0, E4 0 } C_DIS
LIN{ E6POS: X 724.8609, Y 51.3368, Z -174.0150, A 0, B 90, C 0, E1 0, E2 0, E3 0, E4 0 } C_DIS
LIN{ E6POS: X 724.9042, Y 51.4581, Z -174.0150, A 0, B 90, C 0, E1 0, E2 0, E3 0, E4 0 } C_DIS
LIN{ E6POS: X 724.9042, Y 51.4581, Z -174.0150, A 0, B 90, C 0, E1 0, E2 0, E3 0, E4 0 } C_DIS
LIN{ E6POS: X 725.8689, Y 51.1947, Z -174.0150, A 0, B 90, C 0, E1 0, E2 0, E3 0, E4 0 } C_DIS
LIN{ E6POS: X 726.8336, Y 50.9314, Z -174.0150, A 0, B 90, C 0, E1 0, E2 0, E3 0, E4 0 } C_DIS
LIN{ E6POS: X 727.7983, Y 50.6680, Z -174.0150, A 0, B 90, C 0, E1 0, E2 0, E3 0, E4 0 } C_DIS
LIN{ E6POS: X 727.8456, Y 50.6551, Z -174.0150, A 0, B 90, C 0, E1 0, E2 0, E3 0, E4 0 } C_DIS
LIN{ E6POS: X 727.8456, Y 50.6551, Z -174.0150, A 0, B 90, C 0, E1 0, E2 0, E3 0, E4 0 } C_DIS
LIN{ E6POS: X 728.8002, Y 50.3571, Z -174.0150, A 0, B 90, C 0, E1 0, E2 0, E3 0, E4 0 } C_DIS
LIN{ E6POS: X 729.7548, Y 50.0591, Z -174.0150, A 0, B 90, C 0, E1 0, E2 0, E3 0, E4 0 } C_DIS
LIN{ E6POS: X 730.7093, Y 49.7611, Z -174.0150, A 0, B 90, C 0, E1 0, E2 0, E3 0, E4 0 } C_DIS
LIN{ E6POS: X 731.6639, Y 49.4631, Z -174.0150, A 0, B 90, C 0, E1 0, E2 0, E3 0, E4 0 } C_DIS
LIN{ E6POS: X 732.5297, Y 49.1928, Z -174.0150, A 0, B 90, C 0, E1 0, E2 0, E3 0, E4 0 } C_DIS
LIN{ E6POS: X 732.5297, Y 49.1928, Z -174.0150, A 0, B 90, C 0, E1 0, E2 0, E3 0, E4 0 } C_DIS
LIN{ E6POS: X 733.4825, Y 48.8894, Z -174.0150, A 0, B 90, C 0, E1 0, E2 0, E3 0, E4 0 } C_DIS
LIN{ E6POS: X 734.4354, Y 48.5861, Z -174.0150, A 0, B 90, C 0, E1 0, E2 0, E3 0, E4 0 } C_DIS
LIN{ E6POS: X 735.3883, Y 48.2827, Z -174.0150, A 0, B 90, C 0, E1 0, E2 0, E3 0, E4 0 } C_DIS
LIN{ E6POS: X 736.3412, Y 47.9794, Z -174.0150, A 0, B 90, C 0, E1 0, E2 0, E3 0, E4 0 } C_DIS
LIN{ E6POS: X 737.2941, Y 47.6760, Z -174.0150, A 0, B 90, C 0, E1 0, E2 0, E3 0, E4 0 } C_DIS
LIN{ E6POS: X 738.2469, Y 47.3726, Z -174.0150, A 0, B 90, C 0, E1 0, E2 0, E3 0, E4 0 } C_DIS
LIN{ E6POS: X 739.1998, Y 47.0693, Z -174.0150, A 0, B 90, C 0, E1 0, E2 0, E3 0, E4 0 } C_DIS
LIN{ E6POS: X 740.1527, Y 46.7659, Z -174.0150, A 0, B 90, C 0, E1 0, E2 0, E3 0, E4 0 } C_DIS
LIN{ E6POS: X 740.3308, Y 46.7092, Z -174.0150, A 0, B 90, C 0, E1 0, E2 0, E3 0, E4 0 } C_DIS
LIN{ E6POS: X 740.3308, Y 46.7092, Z -174.0150, A 0, B 90, C 0, E1 0, E2 0, E3 0, E4 0 } C_DIS
LIN{ E6POS: X 741.2878, Y 46.4193, Z -174.0150, A 0, B 90, C 0, E1 0, E2 0, E3 0, E4 0 } C_DIS
LIN{ E6POS: X 742.2449, Y 46.1294, Z -174.0150, A 0, B 90, C 0, E1 0, E2 0, E3 0, E4 0 } C_DIS
LIN{ E6POS: X 743.2019, Y 45.8395, Z -174.0150, A 0, B 90, C 0, E1 0, E2 0, E3 0, E4 0 } C_DIS
LIN{ E6POS: X 744.1589, Y 45.5495, Z -174.0150, A 0, B 90, C 0, E1 0, E2 0, E3 0, E4 0 } C_DIS
LIN{ E6POS: X 745.1160, Y 45.2596, Z -174.0150, A 0, B 90, C 0, E1 0, E2 0, E3 0, E4 0 } C_DIS
LIN{ E6POS: X 746.0730, Y 44.9697, Z -174.0150, A 0, B 90, C 0, E1 0, E2 0, E3 0, E4 0 } C_DIS
LIN{ E6POS: X 747.0301, Y 44.6798, Z -174.0150, A 0, B 90, C 0, E1 0, E2 0, E3 0, E4 0 } C_DIS
LIN{ E6POS: X 747.9871, Y 44.3898, Z -174.0150, A 0, B 90, C 0, E1 0, E2 0, E3 0, E4 0 } C_DIS
LIN{ E6POS: X 748.9442, Y 44.0999, Z -174.0150, A 0, B 90, C 0, E1 0, E2 0, E3 0, E4 0 } C_DIS
LIN{ E6POS: X 749.9012, Y 43.8100, Z -174.0150, A 0, B 90, C 0, E1 0, E2 0, E3 0, E4 0 } C_DIS
LIN{ E6POS: X 750.0673, Y 43.7597, Z -174.0150, A 0, B 90, C 0, E1 0, E2 0, E3 0, E4 0 } C_DIS
LIN{ E6POS: X 750.0673, Y 43.7597, Z -174.0150, A 0, B 90, C 0, E1 0, E2 0, E3 0, E4 0 } C_DIS
LIN{ E6POS: X 751.0321, Y 43.4967, Z -174.0150, A 0, B 90, C 0, E1 0, E2 0, E3 0, E4 0 } C_DIS
LIN{ E6POS: X 751.9969, Y 43.2337, Z -174.0150, A 0, B 90, C 0, E1 0, E2 0, E3 0, E4 0 } C_DIS
LIN{ E6POS: X 752.9617, Y 42.9708, Z -174.0150, A 0, B 90, C 0, E1 0, E2 0, E3 0, E4 0 } C_DIS
LIN{ E6POS: X 753.9265, Y 42.7078, Z -174.0150, A 0, B 90, C 0, E1 0, E2 0, E3 0, E4 0 } C_DIS
LIN{ E6POS: X 754.8913, Y 42.4448, Z -174.0150, A 0, B 90, C 0, E1 0, E2 0, E3 0, E4 0 } C_DIS
LIN{ E6POS: X 755.8561, Y 42.1818, Z -174.0150, A 0, B 90, C 0, E1 0, E2 0, E3 0, E4 0 } C_DIS
LIN{ E6POS: X 756.8209, Y 41.9189, Z -174.0150, A 0, B 90, C 0, E1 0, E2 0, E3 0, E4 0 } C_DIS
LIN{ E6POS: X 757.7857, Y 41.6559, Z -174.0150, A 0, B 90, C 0, E1 0, E2 0, E3 0, E4 0 } C_DIS
LIN{ E6POS: X 758.7505, Y 41.3929, Z -174.0150, A 0, B 90, C 0, E1 0, E2 0, E3 0, E4 0 } C_DIS
LIN{ E6POS: X 759.7153, Y 41.1300, Z -174.0150, A 0, B 90, C 0, E1 0, E2 0, E3 0, E4 0 } C_DIS
LIN{ E6POS: X 760.5580, Y 40.9003, Z -174.0150, A 0, B 90, C 0, E1 0, E2 0, E3 0, E4 0 } C_DIS
LIN{ E6POS: X 760.5580, Y 40.9003, Z -174.0150, A 0, B 90, C 0, E1 0, E2 0, E3 0, E4 0 } C_DIS
LIN{ E6POS: X 761.5347, Y 40.6854, Z -174.0150, A 0, B 90, C 0, E1 0, E2 0, E3 0, E4 0 } C_DIS
LIN{ E6POS: X 762.5113, Y 40.4705, Z -174.0150, A 0, B 90, C 0, E1 0, E2 0, E3 0, E4 0 } C_DIS
LIN{ E6POS: X 763.4879, Y 40.2556, Z -174.0150, A 0, B 90, C 0, E1 0, E2 0, E3 0, E4 0 } C_DIS
LIN{ E6POS: X 764.4646, Y 40.0407, Z -174.0150, A 0, B 90, C 0, E1 0, E2 0, E3 0, E4 0 } C_DIS
LIN{ E6POS: X 765.4412, Y 39.8258, Z -174.0150, A 0, B 90, C 0, E1 0, E2 0, E3 0, E4 0 } C_DIS
LIN{ E6POS: X 766.4179, Y 39.6110, Z -174.0150, A 0, B 90, C 0, E1 0, E2 0, E3 0, E4 0 } C_DIS
LIN{ E6POS: X 767.3945, Y 39.3961, Z -174.0150, A 0, B 90, C 0, E1 0, E2 0, E3 0, E4 0 } C_DIS
LIN{ E6POS: X 768.3711, Y 39.1812, Z -174.0150, A 0, B 90, C 0, E1 0, E2 0, E3 0, E4 0 } C_DIS
LIN{ E6POS: X 769.3478, Y 38.9663, Z -174.0150, A 0, B 90, C 0, E1 0, E2 0, E3 0, E4 0 } C_DIS
LIN{ E6POS: X 770.3244, Y 38.7514, Z -174.0150, A 0, B 90, C 0, E1 0, E2 0, E3 0, E4 0 } C_DIS
LIN{ E6POS: X 770.6222, Y 38.6859, Z -174.0150, A 0, B 90, C 0, E1 0, E2 0, E3 0, E4 0 } C_DIS
LIN{ E6POS: X 770.6222, Y 38.6859, Z -174.0150, A 0, B 90, C 0, E1 0, E2 0, E3 0, E4 0 } C_DIS
LIN{ E6POS: X 771.6150, Y 38.5666, Z -174.0150, A 0, B 90, C 0, E1 0, E2 0, E3 0, E4 0 } C_DIS
LIN{ E6POS: X 772.6079, Y 38.4474, Z -174.0150, A 0, B 90, C 0, E1 0, E2 0, E3 0, E4 0 } C_DIS
LIN{ E6POS: X 773.6008, Y 38.3281, Z -174.0150, A 0, B 90, C 0, E1 0, E2 0, E3 0, E4 0 } C_DIS
LIN{ E6POS: X 774.5936, Y 38.2088, Z -174.0150, A 0, B 90, C 0, E1 0, E2 0, E3 0, E4 0 } C_DIS
LIN{ E6POS: X 775.5865, Y 38.0895, Z -174.0150, A 0, B 90, C 0, E1 0, E2 0, E3 0, E4 0 } C_DIS
LIN{ E6POS: X 776.5793, Y 37.9703, Z -174.0150, A 0, B 90, C 0, E1 0, E2 0, E3 0, E4 0 } C_DIS
LIN{ E6POS: X 777.5722, Y 37.8510, Z -174.0150, A 0, B 90, C 0, E1 0, E2 0, E3 0, E4 0 } C_DIS
LIN{ E6POS: X 778.5651, Y 37.7317, Z -174.0150, A 0, B 90, C 0, E1 0, E2 0, E3 0, E4 0 } C_DIS
LIN{ E6POS: X 779.0769, Y 37.6702, Z -174.0150, A 0, B 90, C 0, E1 0, E2 0, E3 0, E4 0 } C_DIS
LIN{ E6POS: X 779.0769, Y 37.6702, Z -174.0150, A 0, B 90, C 0, E1 0, E2 0, E3 0, E4 0 } C_DIS
LIN{ E6POS: X 780.0767, Y 37.6544, Z -174.0150, A 0, B 90, C 0, E1 0, E2 0, E3 0, E4 0 } C_DIS
LIN{ E6POS: X 781.0766, Y 37.6385, Z -174.0150, A 0, B 90, C 0, E1 0, E2 0, E3 0, E4 0 } C_DIS
LIN{ E6POS: X 782.0765, Y 37.6227, Z -174.0150, A 0, B 90, C 0, E1 0, E2 0, E3 0, E4 0 } C_DIS
LIN{ E6POS: X 783.0764, Y 37.6069, Z -174.0150, A 0, B 90, C 0, E1 0, E2 0, E3 0, E4 0 } C_DIS
LIN{ E6POS: X 784.0762, Y 37.5910, Z -174.0150, A 0, B 90, C 0, E1 0, E2 0, E3 0, E4 0 } C_DIS
LIN{ E6POS: X 785.0761, Y 37.5752, Z -174.0150, A 0, B 90, C 0, E1 0, E2 0, E3 0, E4 0 } C_DIS
LIN{ E6POS: X 786.0760, Y 37.5593, Z -174.0150, A 0, B 90, C 0, E1 0, E2 0, E3 0, E4 0 } C_DIS
LIN{ E6POS: X 786.3249, Y 37.5554, Z -174.0150, A 0, B 90, C 0, E1 0, E2 0, E3 0, E4 0 } C_DIS
LIN{ E6POS: X 786.3249, Y 37.5554, Z -174.0150, A 0, B 90, C 0, E1 0, E2 0, E3 0, E4 0 } C_DIS
LIN{ E6POS: X 787.3221, Y 37.6305, Z -174.0150, A 0, B 90, C 0, E1 0, E2 0, E3 0, E4 0 } C_DIS
LIN{ E6POS: X 788.3193, Y 37.7057, Z -174.0150, A 0, B 90, C 0, E1 0, E2 0, E3 0, E4 0 } C_DIS
LIN{ E6POS: X 789.3164, Y 37.7808, Z -174.0150, A 0, B 90, C 0, E1 0, E2 0, E3 0, E4 0 } C_DIS
LIN{ E6POS: X 790.3136, Y 37.8559, Z -174.0150, A 0, B 90, C 0, E1 0, E2 0, E3 0, E4 0 } C_DIS
LIN{ E6POS: X 791.3108, Y 37.9311, Z -174.0150, A 0, B 90, C 0, E1 0, E2 0, E3 0, E4 0 } C_DIS
LIN{ E6POS: X 792.3080, Y 38.0062, Z -174.0150, A 0, B 90, C 0, E1 0, E2 0, E3 0, E4 0 } C_DIS
LIN{ E6POS: X 792.7685, Y 38.0409, Z -174.0150, A 0, B 90, C 0, E1 0, E2 0, E3 0, E4 0 } C_DIS
LIN{ E6POS: X 792.7685, Y 38.0409, Z -174.0150, A 0, B 90, C 0, E1 0, E2 0, E3 0, E4 0 } C_DIS
LIN{ E6POS: X 793.7601, Y 38.1698, Z -174.0150, A 0, B 90, C 0, E1 0, E2 0, E3 0, E4 0 } C_DIS
LIN{ E6POS: X 794.7518, Y 38.2986, Z -174.0150, A 0, B 90, C 0, E1 0, E2 0, E3 0, E4 0 } C_DIS
LIN{ E6POS: X 795.7435, Y 38.4275, Z -174.0150, A 0, B 90, C 0, E1 0, E2 0, E3 0, E4 0 } C_DIS
LIN{ E6POS: X 796.7351, Y 38.5564, Z -174.0150, A 0, B 90, C 0, E1 0, E2 0, E3 0, E4 0 } C_DIS
LIN{ E6POS: X 797.7268, Y 38.6853, Z -174.0150, A 0, B 90, C 0, E1 0, E2 0, E3 0, E4 0 } C_DIS
LIN{ E6POS: X 798.7184, Y 38.8142, Z -174.0150, A 0, B 90, C 0, E1 0, E2 0, E3 0, E4 0 } C_DIS
LIN{ E6POS: X 798.8097, Y 38.8260, Z -174.0150, A 0, B 90, C 0, E1 0, E2 0, E3 0, E4 0 } C_DIS
LIN{ E6POS: X 798.8097, Y 38.8260, Z -174.0150, A 0, B 90, C 0, E1 0, E2 0, E3 0, E4 0 } C_DIS
LIN{ E6POS: X 798.7068, Y 37.8313, Z -174.0150, A 0, B 90, C 0, E1 0, E2 0, E3 0, E4 0 } C_DIS
LIN{ E6POS: X 798.6040, Y 36.8366, Z -174.0150, A 0, B 90, C 0, E1 0, E2 0, E3 0, E4 0 } C_DIS
LIN{ E6POS: X 798.5012, Y 35.8419, Z -174.0150, A 0, B 90, C 0, E1 0, E2 0, E3 0, E4 0 } C_DIS
LIN{ E6POS: X 798.3983, Y 34.8472, Z -174.0150, A 0, B 90, C 0, E1 0, E2 0, E3 0, E4 0 } C_DIS
LIN{ E6POS: X 798.2955, Y 33.8525, Z -174.0150, A 0, B 90, C 0, E1 0, E2 0, E3 0, E4 0 } C_DIS
LIN{ E6POS: X 798.1927, Y 32.8578, Z -174.0150, A 0, B 90, C 0, E1 0, E2 0, E3 0, E4 0 } C_DIS
LIN{ E6POS: X 798.0898, Y 31.8631, Z -174.0150, A 0, B 90, C 0, E1 0, E2 0, E3 0, E4 0 } C_DIS
LIN{ E6POS: X 797.9870, Y 30.8684, Z -174.0150, A 0, B 90, C 0, E1 0, E2 0, E3 0, E4 0 } C_DIS
LIN{ E6POS: X 797.8842, Y 29.8737, Z -174.0150, A 0, B 90, C 0, E1 0, E2 0, E3 0, E4 0 } C_DIS
LIN{ E6POS: X 797.7813, Y 28.8790, Z -174.0150, A 0, B 90, C 0, E1 0, E2 0, E3 0, E4 0 } C_DIS
LIN{ E6POS: X 797.6785, Y 27.8843, Z -174.0150, A 0, B 90, C 0, E1 0, E2 0, E3 0, E4 0 } C_DIS
LIN{ E6POS: X 797.5757, Y 26.8896, Z -174.0150, A 0, B 90, C 0, E1 0, E2 0, E3 0, E4 0 } C_DIS
LIN{ E6POS: X 797.4728, Y 25.8949, Z -174.0150, A 0, B 90, C 0, E1 0, E2 0, E3 0, E4 0 } C_DIS
LIN{ E6POS: X 797.3700, Y 24.9002, Z -174.0150, A 0, B 90, C 0, E1 0, E2 0, E3 0, E4 0 } C_DIS
LIN{ E6POS: X 797.2672, Y 23.9055, Z -174.0150, A 0, B 90, C 0, E1 0, E2 0, E3 0, E4 0 } C_DIS
LIN{ E6POS: X 797.1643, Y 22.9108, Z -174.0150, A 0, B 90, C 0, E1 0, E2 0, E3 0, E4 0 } C_DIS
LIN{ E6POS: X 797.1224, Y 22.5051, Z -174.0150, A 0, B 90, C 0, E1 0, E2 0, E3 0, E4 0 } C_DIS
LIN{ E6POS: X 797.1224, Y 22.5051, Z -174.0150, A 0, B 90, C 0, E1 0, E2 0, E3 0, E4 0 } C_DIS
LIN{ E6POS: X 797.0002, Y 21.5126, Z -174.0150, A 0, B 90, C 0, E1 0, E2 0, E3 0, E4 0 } C_DIS
LIN{ E6POS: X 796.8780, Y 20.5201, Z -174.0150, A 0, B 90, C 0, E1 0, E2 0, E3 0, E4 0 } C_DIS
LIN{ E6POS: X 796.7559, Y 19.5276, Z -174.0150, A 0, B 90, C 0, E1 0, E2 0, E3 0, E4 0 } C_DIS
LIN{ E6POS: X 796.6337, Y 18.5351, Z -174.0150, A 0, B 90, C 0, E1 0, E2 0, E3 0, E4 0 } C_DIS
LIN{ E6POS: X 796.5115, Y 17.5426, Z -174.0150, A 0, B 90, C 0, E1 0, E2 0, E3 0, E4 0 } C_DIS
LIN{ E6POS: X 796.3893, Y 16.5500, Z -174.0150, A 0, B 90, C 0, E1 0, E2 0, E3 0, E4 0 } C_DIS
LIN{ E6POS: X 796.2672, Y 15.5575, Z -174.0150, A 0, B 90, C 0, E1 0, E2 0, E3 0, E4 0 } C_DIS
LIN{ E6POS: X 796.1450, Y 14.5650, Z -174.0150, A 0, B 90, C 0, E1 0, E2 0, E3 0, E4 0 } C_DIS
LIN{ E6POS: X 796.0228, Y 13.5725, Z -174.0150, A 0, B 90, C 0, E1 0, E2 0, E3 0, E4 0 } C_DIS
LIN{ E6POS: X 795.9006, Y 12.5800, Z -174.0150, A 0, B 90, C 0, E1 0, E2 0, E3 0, E4 0 } C_DIS
LIN{ E6POS: X 795.7785, Y 11.5875, Z -174.0150, A 0, B 90, C 0, E1 0, E2 0, E3 0, E4 0 } C_DIS
LIN{ E6POS: X 795.6563, Y 10.5950, Z -174.0150, A 0, B 90, C 0, E1 0, E2 0, E3 0, E4 0 } C_DIS
LIN{ E6POS: X 795.5341, Y 9.6025, Z -174.0150, A 0, B 90, C 0, E1 0, E2 0, E3 0, E4 0 } C_DIS
LIN{ E6POS: X 795.4119, Y 8.6100, Z -174.0150, A 0, B 90, C 0, E1 0, E2 0, E3 0, E4 0 } C_DIS
LIN{ E6POS: X 795.2897, Y 7.6175, Z -174.0150, A 0, B 90, C 0, E1 0, E2 0, E3 0, E4 0 } C_DIS
LIN{ E6POS: X 795.2562, Y 7.3452, Z -174.0150, A 0, B 90, C 0, E1 0, E2 0, E3 0, E4 0 } C_DIS
LIN{ E6POS: X 795.2562, Y 7.3452, Z -174.0150, A 0, B 90, C 0, E1 0, E2 0, E3 0, E4 0 } C_DIS
LIN{ E6POS: X 795.0854, Y 6.3599, Z -174.0150, A 0, B 90, C 0, E1 0, E2 0, E3 0, E4 0 } C_DIS
LIN{ E6POS: X 794.9146, Y 5.3746, Z -174.0150, A 0, B 90, C 0, E1 0, E2 0, E3 0, E4 0 } C_DIS
LIN{ E6POS: X 794.7438, Y 4.3893, Z -174.0150, A 0, B 90, C 0, E1 0, E2 0, E3 0, E4 0 } C_DIS
LIN{ E6POS: X 794.5730, Y 3.4040, Z -174.0150, A 0, B 90, C 0, E1 0, E2 0, E3 0, E4 0 } C_DIS
LIN{ E6POS: X 794.4021, Y 2.4187, Z -174.0150, A 0, B 90, C 0, E1 0, E2 0, E3 0, E4 0 } C_DIS
LIN{ E6POS: X 794.2313, Y 1.4334, Z -174.0150, A 0, B 90, C 0, E1 0, E2 0, E3 0, E4 0 } C_DIS
LIN{ E6POS: X 794.0605, Y 0.4481, Z -174.0150, A 0, B 90, C 0, E1 0, E2 0, E3 0, E4 0 } C_DIS
LIN{ E6POS: X 793.8897, Y -0.5372, Z -174.0150, A 0, B 90, C 0, E1 0, E2 0, E3 0, E4 0 } C_DIS
LIN{ E6POS: X 793.7189, Y -1.5225, Z -174.0150, A 0, B 90, C 0, E1 0, E2 0, E3 0, E4 0 } C_DIS
LIN{ E6POS: X 793.5481, Y -2.5078, Z -174.0150, A 0, B 90, C 0, E1 0, E2 0, E3 0, E4 0 } C_DIS
LIN{ E6POS: X 793.3772, Y -3.4931, Z -174.0150, A 0, B 90, C 0, E1 0, E2 0, E3 0, E4 0 } C_DIS
LIN{ E6POS: X 793.2064, Y -4.4784, Z -174.0150, A 0, B 90, C 0, E1 0, E2 0, E3 0, E4 0 } C_DIS
LIN{ E6POS: X 793.0356, Y -5.4637, Z -174.0150, A 0, B 90, C 0, E1 0, E2 0, E3 0, E4 0 } C_DIS
LIN{ E6POS: X 793.0310, Y -5.4900, Z -172.0150, A 0, B 90, C 0, E1 0, E2 0, E3 0, E4 0 } C_DIS
LIN{ E6POS: X 792.8100, Y -6.2379, Z -172.0150, A 0, B 90, C 0, E1 0, E2 0, E3 0, E4 0 } C_DIS
LIN{ E6POS: X 792.5266, Y -7.1969, Z -172.0150, A 0, B 90, C 0, E1 0, E2 0, E3 0, E4 0 } C_DIS
LIN{ E6POS: X 792.2432, Y -8.1559, Z -172.0150, A 0, B 90, C 0, E1 0, E2 0, E3 0, E4 0 } C_DIS
LIN{ E6POS: X 791.9597, Y -9.1149, Z -172.0150, A 0, B 90, C 0, E1 0, E2 0, E3 0, E4 0 } C_DIS
LIN{ E6POS: X 791.6763, Y -10.0739, Z -172.0150, A 0, B 90, C 0, E1 0, E2 0, E3 0, E4 0 } C_DIS
LIN{ E6POS: X 791.3929, Y -11.0329, Z -172.0150, A 0, B 90, C 0, E1 0, E2 0, E3 0, E4 0 } C_DIS
LIN{ E6POS: X 791.1095, Y -11.9919, Z -172.0150, A 0, B 90, C 0, E1 0, E2 0, E3 0, E4 0 } C_DIS
LIN{ E6POS: X 790.8261, Y -12.9509, Z -172.0150, A 0, B 90, C 0, E1 0, E2 0, E3 0, E4 0 } C_DIS
LIN{ E6POS: X 790.5426, Y -13.9099, Z -172.0150, A 0, B 90, C 0, E1 0, E2 0, E3 0, E4 0 } C_DIS
LIN{ E6POS: X 790.2681, Y -14.8387, Z -172.0150, A 0, B 90, C 0, E1 0, E2 0, E3 0, E4 0 } C_DIS
LIN{ E6POS: X 789.9898, Y -15.2149, Z -172.0150, A 0, B 90, C 0, E1 0, E2 0, E3 0, E4 0 } C_DIS
LIN{ E6POS: X 789.3949, Y -16.0187, Z -172.0150, A 0, B 90, C 0, E1 0, E2 0, E3 0, E4 0 } C_DIS
LIN{ E6POS: X 788.8000, Y -16.8226, Z -172.0150, A 0, B 90, C 0, E1 0, E2 0, E3 0, E4 0 } C_DIS
LIN{ E6POS: X 788.2052, Y -17.6264, Z -172.0150, A 0, B 90, C 0, E1 0, E2 0, E3 0, E4 0 } C_DIS
LIN{ E6POS: X 787.6103, Y -18.4302, Z -172.0150, A 0, B 90, C 0, E1 0, E2 0, E3 0, E4 0 } C_DIS
LIN{ E6POS: X 787.0154, Y -19.2340, Z -172.0150, A 0, B 90, C 0, E1 0, E2 0, E3 0, E4 0 } C_DIS
LIN{ E6POS: X 786.7884, Y -19.5408, Z -172.0150, A 0, B 90, C 0, E1 0, E2 0, E3 0, E4 0 } C_DIS
LIN{ E6POS: X 786.4437, Y -19.6480, Z -172.0150, A 0, B 90, C 0, E1 0, E2 0, E3 0, E4 0 } C_DIS
LIN{ E6POS: X 785.4902, Y -19.9492, Z -172.0150, A 0, B 90, C 0, E1 0, E2 0, E3 0, E4 0 } C_DIS
LIN{ E6POS: X 784.5366, Y -20.2503, Z -172.0150, A 0, B 90, C 0, E1 0, E2 0, E3 0, E4 0 } C_DIS
LIN{ E6POS: X 783.5830, Y -20.5515, Z -172.0150, A 0, B 90, C 0, E1 0, E2 0, E3 0, E4 0 } C_DIS
LIN{ E6POS: X 782.6295, Y -20.8527, Z -172.0150, A 0, B 90, C 0, E1 0, E2 0, E3 0, E4 0 } C_DIS
LIN{ E6POS: X 782.5340, Y -20.8828, Z -172.0150, A 0, B 90, C 0, E1 0, E2 0, E3 0, E4 0 } C_DIS
LIN{ E6POS: X 781.5441, Y -20.7409, Z -172.0150, A 0, B 90, C 0, E1 0, E2 0, E3 0, E4 0 } C_DIS
LIN{ E6POS: X 780.5542, Y -20.5990, Z -172.0150, A 0, B 90, C 0, E1 0, E2 0, E3 0, E4 0 } C_DIS
LIN{ E6POS: X 779.5644, Y -20.4571, Z -172.0150, A 0, B 90, C 0, E1 0, E2 0, E3 0, E4 0 } C_DIS
LIN{ E6POS: X 778.5745, Y -20.3152, Z -172.0150, A 0, B 90, C 0, E1 0, E2 0, E3 0, E4 0 } C_DIS
LIN{ E6POS: X 777.8687, Y -20.2140, Z -172.0150, A 0, B 90, C 0, E1 0, E2 0, E3 0, E4 0 } C_DIS
LIN{ E6POS: X 777.4490, Y -20.1555, Z -172.0150, A 0, B 90, C 0, E1 0, E2 0, E3 0, E4 0 } C_DIS
LIN{ E6POS: X 776.4797, Y -19.9096, Z -172.0150, A 0, B 90, C 0, E1 0, E2 0, E3 0, E4 0 } C_DIS
LIN{ E6POS: X 775.5104, Y -19.6637, Z -172.0150, A 0, B 90, C 0, E1 0, E2 0, E3 0, E4 0 } C_DIS
LIN{ E6POS: X 774.5411, Y -19.4178, Z -172.0150, A 0, B 90, C 0, E1 0, E2 0, E3 0, E4 0 } C_DIS
LIN{ E6POS: X 773.5718, Y -19.1720, Z -172.0150, A 0, B 90, C 0, E1 0, E2 0, E3 0, E4 0 } C_DIS
LIN{ E6POS: X 772.6025, Y -18.9261, Z -172.0150, A 0, B 90, C 0, E1 0, E2 0, E3 0, E4 0 } C_DIS
LIN{ E6POS: X 771.9789, Y -18.7679, Z -172.0150, A 0, B 90, C 0, E1 0, E2 0, E3 0, E4 0 } C_DIS
LIN{ E6POS: X 771.4752, Y -18.6464, Z -172.0150, A 0, B 90, C 0, E1 0, E2 0, E3 0, E4 0 } C_DIS
LIN{ E6POS: X 770.4856, Y -18.5025, Z -172.0150, A 0, B 90, C 0, E1 0, E2 0, E3 0, E4 0 } C_DIS
LIN{ E6POS: X 769.4960, Y -18.3587, Z -172.0150, A 0, B 90, C 0, E1 0, E2 0, E3 0, E4 0 } C_DIS
LIN{ E6POS: X 768.5064, Y -18.2148, Z -172.0150, A 0, B 90, C 0, E1 0, E2 0, E3 0, E4 0 } C_DIS
LIN{ E6POS: X 767.5168, Y -18.0709, Z -172.0150, A 0, B 90, C 0, E1 0, E2 0, E3 0, E4 0 } C_DIS
LIN{ E6POS: X 766.5272, Y -17.9271, Z -172.0150, A 0, B 90, C 0, E1 0, E2 0, E3 0, E4 0 } C_DIS
LIN{ E6POS: X 765.5376, Y -17.7832, Z -172.0150, A 0, B 90, C 0, E1 0, E2 0, E3 0, E4 0 } C_DIS
LIN{ E6POS: X 765.1532, Y -17.7273, Z -172.0150, A 0, B 90, C 0, E1 0, E2 0, E3 0, E4 0 } C_DIS
LIN{ E6POS: X 764.5566, Y -17.6459, Z -172.0150, A 0, B 90, C 0, E1 0, E2 0, E3 0, E4 0 } C_DIS
LIN{ E6POS: X 763.5593, Y -17.5728, Z -172.0150, A 0, B 90, C 0, E1 0, E2 0, E3 0, E4 0 } C_DIS
LIN{ E6POS: X 762.5620, Y -17.4996, Z -172.0150, A 0, B 90, C 0, E1 0, E2 0, E3 0, E4 0 } C_DIS
LIN{ E6POS: X 761.5647, Y -17.4265, Z -172.0150, A 0, B 90, C 0, E1 0, E2 0, E3 0, E4 0 } C_DIS
LIN{ E6POS: X 760.5674, Y -17.3534, Z -172.0150, A 0, B 90, C 0, E1 0, E2 0, E3 0, E4 0 } C_DIS
LIN{ E6POS: X 759.5700, Y -17.2802, Z -172.0150, A 0, B 90, C 0, E1 0, E2 0, E3 0, E4 0 } C_DIS
LIN{ E6POS: X 758.5727, Y -17.2071, Z -172.0150, A 0, B 90, C 0, E1 0, E2 0, E3 0, E4 0 } C_DIS
LIN{ E6POS: X 758.0686, Y -17.1702, Z -172.0150, A 0, B 90, C 0, E1 0, E2 0, E3 0, E4 0 } C_DIS
LIN{ E6POS: X 757.4482, Y -17.1268, Z -172.0150, A 0, B 90, C 0, E1 0, E2 0, E3 0, E4 0 } C_DIS
LIN{ E6POS: X 756.4483, Y -17.1176, Z -172.0150, A 0, B 90, C 0, E1 0, E2 0, E3 0, E4 0 } C_DIS
LIN{ E6POS: X 755.4483, Y -17.1085, Z -172.0150, A 0, B 90, C 0, E1 0, E2 0, E3 0, E4 0 } C_DIS
LIN{ E6POS: X 754.4484, Y -17.0994, Z -172.0150, A 0, B 90, C 0, E1 0, E2 0, E3 0, E4 0 } C_DIS
LIN{ E6POS: X 753.4484, Y -17.0903, Z -172.0150, A 0, B 90, C 0, E1 0, E2 0, E3 0, E4 0 } C_DIS
LIN{ E6POS: X 752.4485, Y -17.0811, Z -172.0150, A 0, B 90, C 0, E1 0, E2 0, E3 0, E4 0 } C_DIS
LIN{ E6POS: X 751.4775, Y -17.0723, Z -172.0150, A 0, B 90, C 0, E1 0, E2 0, E3 0, E4 0 } C_DIS
LIN{ E6POS: X 750.9024, Y -17.0648, Z -172.0150, A 0, B 90, C 0, E1 0, E2 0, E3 0, E4 0 } C_DIS
LIN{ E6POS: X 749.9050, Y -17.1363, Z -172.0150, A 0, B 90, C 0, E1 0, E2 0, E3 0, E4 0 } C_DIS
LIN{ E6POS: X 748.9075, Y -17.2078, Z -172.0150, A 0, B 90, C 0, E1 0, E2 0, E3 0, E4 0 } C_DIS
LIN{ E6POS: X 747.9101, Y -17.2794, Z -172.0150, A 0, B 90, C 0, E1 0, E2 0, E3 0, E4 0 } C_DIS
LIN{ E6POS: X 746.9127, Y -17.3509, Z -172.0150, A 0, B 90, C 0, E1 0, E2 0, E3 0, E4 0 } C_DIS
LIN{ E6POS: X 746.1357, Y -17.4066, Z -172.0150, A 0, B 90, C 0, E1 0, E2 0, E3 0, E4 0 } C_DIS
LIN{ E6POS: X 745.6748, Y -17.4329, Z -172.0150, A 0, B 90, C 0, E1 0, E2 0, E3 0, E4 0 } C_DIS
LIN{ E6POS: X 744.7045, Y -17.6746, Z -172.0150, A 0, B 90, C 0, E1 0, E2 0, E3 0, E4 0 } C_DIS
LIN{ E6POS: X 743.7342, Y -17.9164, Z -172.0150, A 0, B 90, C 0, E1 0, E2 0, E3 0, E4 0 } C_DIS
LIN{ E6POS: X 742.7979, Y -18.1497, Z -172.0150, A 0, B 90, C 0, E1 0, E2 0, E3 0, E4 0 } C_DIS
LIN{ E6POS: X 742.5203, Y -18.2077, Z -172.0150, A 0, B 90, C 0, E1 0, E2 0, E3 0, E4 0 } C_DIS
LIN{ E6POS: X 741.8362, Y -18.9371, Z -172.0150, A 0, B 90, C 0, E1 0, E2 0, E3 0, E4 0 } C_DIS
LIN{ E6POS: X 741.5387, Y -19.2543, Z -172.0150, A 0, B 90, C 0, E1 0, E2 0, E3 0, E4 0 } C_DIS
LIN{ E6POS: X 741.4447, Y -19.3412, Z -172.0150, A 0, B 90, C 0, E1 0, E2 0, E3 0, E4 0 } C_DIS
LIN{ E6POS: X 741.5349, Y -19.4542, Z -172.0150, A 0, B 90, C 0, E1 0, E2 0, E3 0, E4 0 } C_DIS
LIN{ E6POS: X 742.1039, Y -20.2765, Z -172.0150, A 0, B 90, C 0, E1 0, E2 0, E3 0, E4 0 } C_DIS
LIN{ E6POS: X 742.4566, Y -20.7863, Z -172.0150, A 0, B 90, C 0, E1 0, E2 0, E3 0, E4 0 } C_DIS
LIN{ E6POS: X 742.7311, Y -20.9226, Z -172.0150, A 0, B 90, C 0, E1 0, E2 0, E3 0, E4 0 } C_DIS
LIN{ E6POS: X 743.6050, Y -21.4087, Z -172.0150, A 0, B 90, C 0, E1 0, E2 0, E3 0, E4 0 } C_DIS
LIN{ E6POS: X 744.4789, Y -21.8948, Z -172.0150, A 0, B 90, C 0, E1 0, E2 0, E3 0, E4 0 } C_DIS
LIN{ E6POS: X 745.3528, Y -22.3808, Z -172.0150, A 0, B 90, C 0, E1 0, E2 0, E3 0, E4 0 } C_DIS
LIN{ E6POS: X 745.5619, Y -22.4971, Z -172.0150, A 0, B 90, C 0, E1 0, E2 0, E3 0, E4 0 } C_DIS
LIN{ E6POS: X 746.0213, Y -22.6540, Z -172.0150, A 0, B 90, C 0, E1 0, E2 0, E3 0, E4 0 } C_DIS
LIN{ E6POS: X 746.9582, Y -23.0036, Z -172.0150, A 0, B 90, C 0, E1 0, E2 0, E3 0, E4 0 } C_DIS
LIN{ E6POS: X 747.8952, Y -23.3532, Z -172.0150, A 0, B 90, C 0, E1 0, E2 0, E3 0, E4 0 } C_DIS
LIN{ E6POS: X 748.8321, Y -23.7027, Z -172.0150, A 0, B 90, C 0, E1 0, E2 0, E3 0, E4 0 } C_DIS
LIN{ E6POS: X 749.7690, Y -24.0523, Z -172.0150, A 0, B 90, C 0, E1 0, E2 0, E3 0, E4 0 } C_DIS
LIN{ E6POS: X 750.7059, Y -24.4019, Z -172.0150, A 0, B 90, C 0, E1 0, E2 0, E3 0, E4 0 } C_DIS
LIN{ E6POS: X 750.7695, Y -24.4256, Z -172.0150, A 0, B 90, C 0, E1 0, E2 0, E3 0, E4 0 } C_DIS
LIN{ E6POS: X 751.3444, Y -24.5806, Z -172.0150, A 0, B 90, C 0, E1 0, E2 0, E3 0, E4 0 } C_DIS
LIN{ E6POS: X 752.3051, Y -24.8582, Z -172.0150, A 0, B 90, C 0, E1 0, E2 0, E3 0, E4 0 } C_DIS
LIN{ E6POS: X 753.2658, Y -25.1358, Z -172.0150, A 0, B 90, C 0, E1 0, E2 0, E3 0, E4 0 } C_DIS
LIN{ E6POS: X 754.2265, Y -25.4134, Z -172.0150, A 0, B 90, C 0, E1 0, E2 0, E3 0, E4 0 } C_DIS
LIN{ E6POS: X 755.1872, Y -25.6910, Z -172.0150, A 0, B 90, C 0, E1 0, E2 0, E3 0, E4 0 } C_DIS
LIN{ E6POS: X 756.1479, Y -25.9686, Z -172.0150, A 0, B 90, C 0, E1 0, E2 0, E3 0, E4 0 } C_DIS
LIN{ E6POS: X 757.1086, Y -26.2462, Z -172.0150, A 0, B 90, C 0, E1 0, E2 0, E3 0, E4 0 } C_DIS
LIN{ E6POS: X 757.3168, Y -26.3064, Z -172.0150, A 0, B 90, C 0, E1 0, E2 0, E3 0, E4 0 } C_DIS
LIN{ E6POS: X 757.9377, Y -26.4369, Z -172.0150, A 0, B 90, C 0, E1 0, E2 0, E3 0, E4 0 } C_DIS
LIN{ E6POS: X 758.9142, Y -26.6526, Z -172.0150, A 0, B 90, C 0, E1 0, E2 0, E3 0, E4 0 } C_DIS
LIN{ E6POS: X 759.8906, Y -26.8684, Z -172.0150, A 0, B 90, C 0, E1 0, E2 0, E3 0, E4 0 } C_DIS
LIN{ E6POS: X 760.8671, Y -27.0841, Z -172.0150, A 0, B 90, C 0, E1 0, E2 0, E3 0, E4 0 } C_DIS
LIN{ E6POS: X 761.8435, Y -27.2999, Z -172.0150, A 0, B 90, C 0, E1 0, E2 0, E3 0, E4 0 } C_DIS
LIN{ E6POS: X 762.8200, Y -27.5156, Z -172.0150, A 0, B 90, C 0, E1 0, E2 0, E3 0, E4 0 } C_DIS
LIN{ E6POS: X 763.7964, Y -27.7314, Z -172.0150, A 0, B 90, C 0, E1 0, E2 0, E3 0, E4 0 } C_DIS
LIN{ E6POS: X 764.4419, Y -27.8740, Z -172.0150, A 0, B 90, C 0, E1 0, E2 0, E3 0, E4 0 } C_DIS
LIN{ E6POS: X 765.0397, Y -27.9575, Z -172.0150, A 0, B 90, C 0, E1 0, E2 0, E3 0, E4 0 } C_DIS
LIN{ E6POS: X 766.0297, Y -28.0984, Z -172.0150, A 0, B 90, C 0, E1 0, E2 0, E3 0, E4 0 } C_DIS
LIN{ E6POS: X 767.0197, Y -28.2393, Z -172.0150, A 0, B 90, C 0, E1 0, E2 0, E3 0, E4 0 } C_DIS
LIN{ E6POS: X 768.0097, Y -28.3803, Z -172.0150, A 0, B 90, C 0, E1 0, E2 0, E3 0, E4 0 } C_DIS
LIN{ E6POS: X 768.9998, Y -28.5212, Z -172.0150, A 0, B 90, C 0, E1 0, E2 0, E3 0, E4 0 } C_DIS
LIN{ E6POS: X 769.9898, Y -28.6621, Z -172.0150, A 0, B 90, C 0, E1 0, E2 0, E3 0, E4 0 } C_DIS
LIN{ E6POS: X 770.9798, Y -28.8031, Z -172.0150, A 0, B 90, C 0, E1 0, E2 0, E3 0, E4 0 } C_DIS
LIN{ E6POS: X 771.3840, Y -28.8606, Z -172.0150, A 0, B 90, C 0, E1 0, E2 0, E3 0, E4 0 } C_DIS
LIN{ E6POS: X 771.8892, Y -28.8745, Z -172.0150, A 0, B 90, C 0, E1 0, E2 0, E3 0, E4 0 } C_DIS
LIN{ E6POS: X 772.8889, Y -28.8975, Z -172.0150, A 0, B 90, C 0, E1 0, E2 0, E3 0, E4 0 } C_DIS
LIN{ E6POS: X 773.8886, Y -28.9204, Z -172.0150, A 0, B 90, C 0, E1 0, E2 0, E3 0, E4 0 } C_DIS
LIN{ E6POS: X 774.8884, Y -28.9434, Z -172.0150, A 0, B 90, C 0, E1 0, E2 0, E3 0, E4 0 } C_DIS
LIN{ E6POS: X 775.8881, Y -28.9664, Z -172.0150, A 0, B 90, C 0, E1 0, E2 0, E3 0, E4 0 } C_DIS
LIN{ E6POS: X 776.8878, Y -28.9893, Z -172.0150, A 0, B 90, C 0, E1 0, E2 0, E3 0, E4 0 } C_DIS
LIN{ E6POS: X 777.3805, Y -29.0006, Z -172.0150, A 0, B 90, C 0, E1 0, E2 0, E3 0, E4 0 } C_DIS
LIN{ E6POS: X 777.7691, Y -29.0752, Z -172.0150, A 0, B 90, C 0, E1 0, E2 0, E3 0, E4 0 } C_DIS
LIN{ E6POS: X 778.7506, Y -29.2666, Z -172.0150, A 0, B 90, C 0, E1 0, E2 0, E3 0, E4 0 } C_DIS
LIN{ E6POS: X 779.7321, Y -29.4580, Z -172.0150, A 0, B 90, C 0, E1 0, E2 0, E3 0, E4 0 } C_DIS
LIN{ E6POS: X 780.7136, Y -29.6494, Z -172.0150, A 0, B 90, C 0, E1 0, E2 0, E3 0, E4 0 } C_DIS
LIN{ E6POS: X 781.6951, Y -29.8408, Z -172.0150, A 0, B 90, C 0, E1 0, E2 0, E3 0, E4 0 } C_DIS
LIN{ E6POS: X 782.0792, Y -29.9157, Z -172.0150, A 0, B 90, C 0, E1 0, E2 0, E3 0, E4 0 } C_DIS
LIN{ E6POS: X 782.3273, Y -30.1811, Z -172.0150, A 0, B 90, C 0, E1 0, E2 0, E3 0, E4 0 } C_DIS
LIN{ E6POS: X 783.0042, Y -30.9172, Z -172.0150, A 0, B 90, C 0, E1 0, E2 0, E3 0, E4 0 } C_DIS
LIN{ E6POS: X 783.6811, Y -31.6532, Z -172.0150, A 0, B 90, C 0, E1 0, E2 0, E3 0, E4 0 } C_DIS
LIN{ E6POS: X 784.3581, Y -32.3893, Z -172.0150, A 0, B 90, C 0, E1 0, E2 0, E3 0, E4 0 } C_DIS
LIN{ E6POS: X 785.0350, Y -33.1253, Z -172.0150, A 0, B 90, C 0, E1 0, E2 0, E3 0, E4 0 } C_DIS
LIN{ E6POS: X 785.1281, Y -33.2266, Z -172.0150, A 0, B 90, C 0, E1 0, E2 0, E3 0, E4 0 } C_DIS
LIN{ E6POS: X 785.2118, Y -33.8128, Z -172.0150, A 0, B 90, C 0, E1 0, E2 0, E3 0, E4 0 } C_DIS
LIN{ E6POS: X 785.3532, Y -34.8027, Z -172.0150, A 0, B 90, C 0, E1 0, E2 0, E3 0, E4 0 } C_DIS
LIN{ E6POS: X 785.4946, Y -35.7927, Z -172.0150, A 0, B 90, C 0, E1 0, E2 0, E3 0, E4 0 } C_DIS
LIN{ E6POS: X 785.6360, Y -36.7826, Z -172.0150, A 0, B 90, C 0, E1 0, E2 0, E3 0, E4 0 } C_DIS
LIN{ E6POS: X 785.7774, Y -37.7726, Z -172.0150, A 0, B 90, C 0, E1 0, E2 0, E3 0, E4 0 } C_DIS
LIN{ E6POS: X 785.9188, Y -38.7625, Z -172.0150, A 0, B 90, C 0, E1 0, E2 0, E3 0, E4 0 } C_DIS
LIN{ E6POS: X 786.0602, Y -39.7525, Z -172.0150, A 0, B 90, C 0, E1 0, E2 0, E3 0, E4 0 } C_DIS
LIN{ E6POS: X 786.1747, Y -40.5536, Z -172.0150, A 0, B 90, C 0, E1 0, E2 0, E3 0, E4 0 } C_DIS
LIN{ E6POS: X 786.0743, Y -41.5485, Z -172.0150, A 0, B 90, C 0, E1 0, E2 0, E3 0, E4 0 } C_DIS
LIN{ E6POS: X 786.0701, Y -41.5908, Z -172.0150, A 0, B 90, C 0, E1 0, E2 0, E3 0, E4 0 } C_DIS
LIN{ E6POS: X 785.9698, Y -42.5857, Z -172.0150, A 0, B 90, C 0, E1 0, E2 0, E3 0, E4 0 } C_DIS
LIN{ E6POS: X 785.8695, Y -43.5807, Z -172.0150, A 0, B 90, C 0, E1 0, E2 0, E3 0, E4 0 } C_DIS
LIN{ E6POS: X 785.7691, Y -44.5756, Z -172.0150, A 0, B 90, C 0, E1 0, E2 0, E3 0, E4 0 } C_DIS
LIN{ E6POS: X 785.6688, Y -45.5706, Z -172.0150, A 0, B 90, C 0, E1 0, E2 0, E3 0, E4 0 } C_DIS
LIN{ E6POS: X 785.5685, Y -46.5655, Z -172.0150, A 0, B 90, C 0, E1 0, E2 0, E3 0, E4 0 } C_DIS
LIN{ E6POS: X 785.4682, Y -47.5605, Z -172.0150, A 0, B 90, C 0, E1 0, E2 0, E3 0, E4 0 } C_DIS
LIN{ E6POS: X 785.3679, Y -48.5554, Z -172.0150, A 0, B 90, C 0, E1 0, E2 0, E3 0, E4 0 } C_DIS
LIN{ E6POS: X 785.2676, Y -49.5504, Z -172.0150, A 0, B 90, C 0, E1 0, E2 0, E3 0, E4 0 } C_DIS
LIN{ E6POS: X 785.1673, Y -50.5454, Z -172.0150, A 0, B 90, C 0, E1 0, E2 0, E3 0, E4 0 } C_DIS
LIN{ E6POS: X 785.0669, Y -51.5403, Z -172.0150, A 0, B 90, C 0, E1 0, E2 0, E3 0, E4 0 } C_DIS
LIN{ E6POS: X 784.9666, Y -52.5353, Z -172.0150, A 0, B 90, C 0, E1 0, E2 0, E3 0, E4 0 } C_DIS
LIN{ E6POS: X 784.8675, Y -53.5185, Z -172.0150, A 0, B 90, C 0, E1 0, E2 0, E3 0, E4 0 } C_DIS
LIN{ E6POS: X 784.6915, Y -54.5029, Z -172.0150, A 0, B 90, C 0, E1 0, E2 0, E3 0, E4 0 } C_DIS
LIN{ E6POS: X 784.6216, Y -54.8939, Z -172.0150, A 0, B 90, C 0, E1 0, E2 0, E3 0, E4 0 } C_DIS
LIN{ E6POS: X 784.4457, Y -55.8783, Z -172.0150, A 0, B 90, C 0, E1 0, E2 0, E3 0, E4 0 } C_DIS
LIN{ E6POS: X 784.2697, Y -56.8627, Z -172.0150, A 0, B 90, C 0, E1 0, E2 0, E3 0, E4 0 } C_DIS
LIN{ E6POS: X 784.0938, Y -57.8471, Z -172.0150, A 0, B 90, C 0, E1 0, E2 0, E3 0, E4 0 } C_DIS
LIN{ E6POS: X 783.9178, Y -58.8315, Z -172.0150, A 0, B 90, C 0, E1 0, E2 0, E3 0, E4 0 } C_DIS
LIN{ E6POS: X 783.7419, Y -59.8159, Z -172.0150, A 0, B 90, C 0, E1 0, E2 0, E3 0, E4 0 } C_DIS
LIN{ E6POS: X 783.5659, Y -60.8003, Z -172.0150, A 0, B 90, C 0, E1 0, E2 0, E3 0, E4 0 } C_DIS
LIN{ E6POS: X 783.3900, Y -61.7847, Z -172.0150, A 0, B 90, C 0, E1 0, E2 0, E3 0, E4 0 } C_DIS
LIN{ E6POS: X 783.2140, Y -62.7691, Z -172.0150, A 0, B 90, C 0, E1 0, E2 0, E3 0, E4 0 } C_DIS
LIN{ E6POS: X 783.0381, Y -63.7535, Z -172.0150, A 0, B 90, C 0, E1 0, E2 0, E3 0, E4 0 } C_DIS
LIN{ E6POS: X 782.8621, Y -64.7379, Z -172.0150, A 0, B 90, C 0, E1 0, E2 0, E3 0, E4 0 } C_DIS
LIN{ E6POS: X 782.6862, Y -65.7223, Z -172.0150, A 0, B 90, C 0, E1 0, E2 0, E3 0, E4 0 } C_DIS
LIN{ E6POS: X 782.5102, Y -66.7067, Z -172.0150, A 0, B 90, C 0, E1 0, E2 0, E3 0, E4 0 } C_DIS
LIN{ E6POS: X 782.3343, Y -67.6911, Z -172.0150, A 0, B 90, C 0, E1 0, E2 0, E3 0, E4 0 } C_DIS
LIN{ E6POS: X 782.1583, Y -68.6755, Z -172.0150, A 0, B 90, C 0, E1 0, E2 0, E3 0, E4 0 } C_DIS
LIN{ E6POS: X 781.9824, Y -69.6599, Z -172.0150, A 0, B 90, C 0, E1 0, E2 0, E3 0, E4 0 } C_DIS
LIN{ E6POS: X 781.8064, Y -70.6443, Z -172.0150, A 0, B 90, C 0, E1 0, E2 0, E3 0, E4 0 } C_DIS
LIN{ E6POS: X 781.7943, Y -70.7119, Z -172.0150, A 0, B 90, C 0, E1 0, E2 0, E3 0, E4 0 } C_DIS
LIN{ E6POS: X 781.5865, Y -71.6900, Z -172.0150, A 0, B 90, C 0, E1 0, E2 0, E3 0, E4 0 } C_DIS
LIN{ E6POS: X 781.4542, Y -72.3129, Z -172.0150, A 0, B 90, C 0, E1 0, E2 0, E3 0, E4 0 } C_DIS
LIN{ E6POS: X 781.2464, Y -73.2910, Z -172.0150, A 0, B 90, C 0, E1 0, E2 0, E3 0, E4 0 } C_DIS
LIN{ E6POS: X 781.0386, Y -74.2692, Z -172.0150, A 0, B 90, C 0, E1 0, E2 0, E3 0, E4 0 } C_DIS
LIN{ E6POS: X 780.8308, Y -75.2474, Z -172.0150, A 0, B 90, C 0, E1 0, E2 0, E3 0, E4 0 } C_DIS
LIN{ E6POS: X 780.6230, Y -76.2255, Z -172.0150, A 0, B 90, C 0, E1 0, E2 0, E3 0, E4 0 } C_DIS
LIN{ E6POS: X 780.4152, Y -77.2037, Z -172.0150, A 0, B 90, C 0, E1 0, E2 0, E3 0, E4 0 } C_DIS
LIN{ E6POS: X 780.2074, Y -78.1819, Z -172.0150, A 0, B 90, C 0, E1 0, E2 0, E3 0, E4 0 } C_DIS
LIN{ E6POS: X 779.9996, Y -79.1600, Z -172.0150, A 0, B 90, C 0, E1 0, E2 0, E3 0, E4 0 } C_DIS
LIN{ E6POS: X 779.7918, Y -80.1382, Z -172.0150, A 0, B 90, C 0, E1 0, E2 0, E3 0, E4 0 } C_DIS
LIN{ E6POS: X 779.5840, Y -81.1164, Z -172.0150, A 0, B 90, C 0, E1 0, E2 0, E3 0, E4 0 } C_DIS
LIN{ E6POS: X 779.3762, Y -82.0946, Z -172.0150, A 0, B 90, C 0, E1 0, E2 0, E3 0, E4 0 } C_DIS
LIN{ E6POS: X 779.1684, Y -83.0727, Z -172.0150, A 0, B 90, C 0, E1 0, E2 0, E3 0, E4 0 } C_DIS
LIN{ E6POS: X 778.9606, Y -84.0509, Z -172.0150, A 0, B 90, C 0, E1 0, E2 0, E3 0, E4 0 } C_DIS
LIN{ E6POS: X 778.7528, Y -85.0291, Z -172.0150, A 0, B 90, C 0, E1 0, E2 0, E3 0, E4 0 } C_DIS
LIN{ E6POS: X 778.5450, Y -86.0072, Z -172.0150, A 0, B 90, C 0, E1 0, E2 0, E3 0, E4 0 } C_DIS
LIN{ E6POS: X 778.3372, Y -86.9854, Z -172.0150, A 0, B 90, C 0, E1 0, E2 0, E3 0, E4 0 } C_DIS
LIN{ E6POS: X 778.1294, Y -87.9636, Z -172.0150, A 0, B 90, C 0, E1 0, E2 0, E3 0, E4 0 } C_DIS
LIN{ E6POS: X 777.9216, Y -88.9418, Z -172.0150, A 0, B 90, C 0, E1 0, E2 0, E3 0, E4 0 } C_DIS
LIN{ E6POS: X 777.7138, Y -89.9199, Z -172.0150, A 0, B 90, C 0, E1 0, E2 0, E3 0, E4 0 } C_DIS
LIN{ E6POS: X 777.5429, Y -90.7243, Z -172.0150, A 0, B 90, C 0, E1 0, E2 0, E3 0, E4 0 } C_DIS
LIN{ E6POS: X 777.3226, Y -91.6997, Z -172.0150, A 0, B 90, C 0, E1 0, E2 0, E3 0, E4 0 } C_DIS
LIN{ E6POS: X 777.1558, Y -92.4381, Z -172.0150, A 0, B 90, C 0, E1 0, E2 0, E3 0, E4 0 } C_DIS
LIN{ E6POS: X 776.9354, Y -93.4135, Z -172.0150, A 0, B 90, C 0, E1 0, E2 0, E3 0, E4 0 } C_DIS
LIN{ E6POS: X 776.7151, Y -94.3889, Z -172.0150, A 0, B 90, C 0, E1 0, E2 0, E3 0, E4 0 } C_DIS
LIN{ E6POS: X 776.4947, Y -95.3643, Z -172.0150, A 0, B 90, C 0, E1 0, E2 0, E3 0, E4 0 } C_DIS
LIN{ E6POS: X 776.2744, Y -96.3397, Z -172.0150, A 0, B 90, C 0, E1 0, E2 0, E3 0, E4 0 } C_DIS
LIN{ E6POS: X 776.0541, Y -97.3152, Z -172.0150, A 0, B 90, C 0, E1 0, E2 0, E3 0, E4 0 } C_DIS
LIN{ E6POS: X 775.8337, Y -98.2906, Z -172.0150, A 0, B 90, C 0, E1 0, E2 0, E3 0, E4 0 } C_DIS
LIN{ E6POS: X 775.6134, Y -99.2660, Z -172.0150, A 0, B 90, C 0, E1 0, E2 0, E3 0, E4 0 } C_DIS
LIN{ E6POS: X 775.3930, Y -100.2414, Z -172.0150, A 0, B 90, C 0, E1 0, E2 0, E3 0, E4 0 } C_DIS
LIN{ E6POS: X 775.1727, Y -101.2169, Z -172.0150, A 0, B 90, C 0, E1 0, E2 0, E3 0, E4 0 } C_DIS
LIN{ E6POS: X 774.9523, Y -102.1923, Z -172.0150, A 0, B 90, C 0, E1 0, E2 0, E3 0, E4 0 } C_DIS
LIN{ E6POS: X 774.7320, Y -103.1677, Z -172.0150, A 0, B 90, C 0, E1 0, E2 0, E3 0, E4 0 } C_DIS
LIN{ E6POS: X 774.5116, Y -104.1431, Z -172.0150, A 0, B 90, C 0, E1 0, E2 0, E3 0, E4 0 } C_DIS
LIN{ E6POS: X 774.2913, Y -105.1185, Z -172.0150, A 0, B 90, C 0, E1 0, E2 0, E3 0, E4 0 } C_DIS
LIN{ E6POS: X 774.0709, Y -106.0940, Z -172.0150, A 0, B 90, C 0, E1 0, E2 0, E3 0, E4 0 } C_DIS
LIN{ E6POS: X 773.8506, Y -107.0694, Z -172.0150, A 0, B 90, C 0, E1 0, E2 0, E3 0, E4 0 } C_DIS
LIN{ E6POS: X 773.6303, Y -108.0448, Z -172.0150, A 0, B 90, C 0, E1 0, E2 0, E3 0, E4 0 } C_DIS
LIN{ E6POS: X 773.4099, Y -109.0202, Z -172.0150, A 0, B 90, C 0, E1 0, E2 0, E3 0, E4 0 } C_DIS
LIN{ E6POS: X 773.1896, Y -109.9956, Z -172.0150, A 0, B 90, C 0, E1 0, E2 0, E3 0, E4 0 } C_DIS
LIN{ E6POS: X 772.9692, Y -110.9711, Z -172.0150, A 0, B 90, C 0, E1 0, E2 0, E3 0, E4 0 } C_DIS
LIN{ E6POS: X 772.7489, Y -111.9465, Z -172.0150, A 0, B 90, C 0, E1 0, E2 0, E3 0, E4 0 } C_DIS
LIN{ E6POS: X 772.7038, Y -112.1462, Z -172.0150, A 0, B 90, C 0, E1 0, E2 0, E3 0, E4 0 } C_DIS
LIN{ E6POS: X 772.4900, Y -111.9045, Z -172.0150, A 0, B 90, C 0, E1 0, E2 0, E3 0, E4 0 } C_DIS
LIN{ E6POS: X 771.8275, Y -111.1555, Z -172.0150, A 0, B 90, C 0, E1 0, E2 0, E3 0, E4 0 } C_DIS
LIN{ E6POS: X 771.1649, Y -110.4064, Z -172.0150, A 0, B 90, C 0, E1 0, E2 0, E3 0, E4 0 } C_DIS
LIN{ E6POS: X 770.5024, Y -109.6574, Z -172.0150, A 0, B 90, C 0, E1 0, E2 0, E3 0, E4 0 } C_DIS
LIN{ E6POS: X 770.0315, Y -109.1250, Z -172.0150, A 0, B 90, C 0, E1 0, E2 0, E3 0, E4 0 } C_DIS
LIN{ E6POS: X 769.7554, Y -108.8741, Z -172.0150, A 0, B 90, C 0, E1 0, E2 0, E3 0, E4 0 } C_DIS
LIN{ E6POS: X 769.0160, Y -108.2008, Z -172.0150, A 0, B 90, C 0, E1 0, E2 0, E3 0, E4 0 } C_DIS
LIN{ E6POS: X 768.2767, Y -107.5274, Z -172.0150, A 0, B 90, C 0, E1 0, E2 0, E3 0, E4 0 } C_DIS
LIN{ E6POS: X 767.5374, Y -106.8540, Z -172.0150, A 0, B 90, C 0, E1 0, E2 0, E3 0, E4 0 } C_DIS
LIN{ E6POS: X 766.7981, Y -106.1807, Z -172.0150, A 0, B 90, C 0, E1 0, E2 0, E3 0, E4 0 } C_DIS
LIN{ E6POS: X 766.6022, Y -106.0023, Z -172.0150, A 0, B 90, C 0, E1 0, E2 0, E3 0, E4 0 } C_DIS
LIN{ E6POS: X 765.7727, Y -105.4438, Z -172.0150, A 0, B 90, C 0, E1 0, E2 0, E3 0, E4 0 } C_DIS
LIN{ E6POS: X 764.9431, Y -104.8854, Z -172.0150, A 0, B 90, C 0, E1 0, E2 0, E3 0, E4 0 } C_DIS
LIN{ E6POS: X 764.1136, Y -104.3269, Z -172.0150, A 0, B 90, C 0, E1 0, E2 0, E3 0, E4 0 } C_DIS
LIN{ E6POS: X 763.2840, Y -103.7685, Z -172.0150, A 0, B 90, C 0, E1 0, E2 0, E3 0, E4 0 } C_DIS
LIN{ E6POS: X 762.4545, Y -103.2101, Z -172.0150, A 0, B 90, C 0, E1 0, E2 0, E3 0, E4 0 } C_DIS
LIN{ E6POS: X 762.0608, Y -102.9451, Z -172.0150, A 0, B 90, C 0, E1 0, E2 0, E3 0, E4 0 } C_DIS
LIN{ E6POS: X 761.6600, Y -102.6759, Z -172.0150, A 0, B 90, C 0, E1 0, E2 0, E3 0, E4 0 } C_DIS
LIN{ E6POS: X 760.7668, Y -102.2263, Z -172.0150, A 0, B 90, C 0, E1 0, E2 0, E3 0, E4 0 } C_DIS
LIN{ E6POS: X 759.8735, Y -101.7768, Z -172.0150, A 0, B 90, C 0, E1 0, E2 0, E3 0, E4 0 } C_DIS
LIN{ E6POS: X 758.9803, Y -101.3272, Z -172.0150, A 0, B 90, C 0, E1 0, E2 0, E3 0, E4 0 } C_DIS
LIN{ E6POS: X 758.0870, Y -100.8777, Z -172.0150, A 0, B 90, C 0, E1 0, E2 0, E3 0, E4 0 } C_DIS
LIN{ E6POS: X 757.1938, Y -100.4281, Z -172.0150, A 0, B 90, C 0, E1 0, E2 0, E3 0, E4 0 } C_DIS
LIN{ E6POS: X 756.3005, Y -99.9786, Z -172.0150, A 0, B 90, C 0, E1 0, E2 0, E3 0, E4 0 } C_DIS
LIN{ E6POS: X 755.4073, Y -99.5290, Z -172.0150, A 0, B 90, C 0, E1 0, E2 0, E3 0, E4 0 } C_DIS
LIN{ E6POS: X 755.0355, Y -99.3419, Z -172.0150, A 0, B 90, C 0, E1 0, E2 0, E3 0, E4 0 } C_DIS
LIN{ E6POS: X 754.4477, Y -99.0451, Z -172.0150, A 0, B 90, C 0, E1 0, E2 0, E3 0, E4 0 } C_DIS
LIN{ E6POS: X 753.5173, Y -98.6786, Z -172.0150, A 0, B 90, C 0, E1 0, E2 0, E3 0, E4 0 } C_DIS
LIN{ E6POS: X 752.5869, Y -98.3121, Z -172.0150, A 0, B 90, C 0, E1 0, E2 0, E3 0, E4 0 } C_DIS
LIN{ E6POS: X 751.6565, Y -97.9455, Z -172.0150, A 0, B 90, C 0, E1 0, E2 0, E3 0, E4 0 } C_DIS
LIN{ E6POS: X 750.7261, Y -97.5790, Z -172.0150, A 0, B 90, C 0, E1 0, E2 0, E3 0, E4 0 } C_DIS
LIN{ E6POS: X 749.7957, Y -97.2124, Z -172.0150, A 0, B 90, C 0, E1 0, E2 0, E3 0, E4 0 } C_DIS
LIN{ E6POS: X 748.8653, Y -96.8459, Z -172.0150, A 0, B 90, C 0, E1 0, E2 0, E3 0, E4 0 } C_DIS
LIN{ E6POS: X 747.9349, Y -96.4794, Z -172.0150, A 0, B 90, C 0, E1 0, E2 0, E3 0, E4 0 } C_DIS
LIN{ E6POS: X 747.0045, Y -96.1128, Z -172.0150, A 0, B 90, C 0, E1 0, E2 0, E3 0, E4 0 } C_DIS
LIN{ E6POS: X 746.0741, Y -95.7463, Z -172.0150, A 0, B 90, C 0, E1 0, E2 0, E3 0, E4 0 } C_DIS
LIN{ E6POS: X 745.1437, Y -95.3797, Z -172.0150, A 0, B 90, C 0, E1 0, E2 0, E3 0, E4 0 } C_DIS
LIN{ E6POS: X 745.0463, Y -95.3414, Z -172.0150, A 0, B 90, C 0, E1 0, E2 0, E3 0, E4 0 } C_DIS
LIN{ E6POS: X 744.2093, Y -95.0081, Z -172.0150, A 0, B 90, C 0, E1 0, E2 0, E3 0, E4 0 } C_DIS
LIN{ E6POS: X 743.2662, Y -94.6754, Z -172.0150, A 0, B 90, C 0, E1 0, E2 0, E3 0, E4 0 } C_DIS
LIN{ E6POS: X 742.3232, Y -94.3427, Z -172.0150, A 0, B 90, C 0, E1 0, E2 0, E3 0, E4 0 } C_DIS
LIN{ E6POS: X 741.3802, Y -94.0099, Z -172.0150, A 0, B 90, C 0, E1 0, E2 0, E3 0, E4 0 } C_DIS
LIN{ E6POS: X 740.4372, Y -93.6772, Z -172.0150, A 0, B 90, C 0, E1 0, E2 0, E3 0, E4 0 } C_DIS
LIN{ E6POS: X 739.4941, Y -93.3445, Z -172.0150, A 0, B 90, C 0, E1 0, E2 0, E3 0, E4 0 } C_DIS
LIN{ E6POS: X 738.5511, Y -93.0118, Z -172.0150, A 0, B 90, C 0, E1 0, E2 0, E3 0, E4 0 } C_DIS
LIN{ E6POS: X 737.6081, Y -92.6791, Z -172.0150, A 0, B 90, C 0, E1 0, E2 0, E3 0, E4 0 } C_DIS
LIN{ E6POS: X 736.6650, Y -92.3464, Z -172.0150, A 0, B 90, C 0, E1 0, E2 0, E3 0, E4 0 } C_DIS
LIN{ E6POS: X 735.7220, Y -92.0137, Z -172.0150, A 0, B 90, C 0, E1 0, E2 0, E3 0, E4 0 } C_DIS
LIN{ E6POS: X 734.7790, Y -91.6809, Z -172.0150, A 0, B 90, C 0, E1 0, E2 0, E3 0, E4 0 } C_DIS
LIN{ E6POS: X 733.8360, Y -91.3482, Z -172.0150, A 0, B 90, C 0, E1 0, E2 0, E3 0, E4 0 } C_DIS
LIN{ E6POS: X 733.5869, Y -91.2603, Z -172.0150, A 0, B 90, C 0, E1 0, E2 0, E3 0, E4 0 } C_DIS
LIN{ E6POS: X 732.6452, Y -90.9238, Z -172.0150, A 0, B 90, C 0, E1 0, E2 0, E3 0, E4 0 } C_DIS
LIN{ E6POS: X 732.6395, Y -90.9217, Z -172.0150, A 0, B 90, C 0, E1 0, E2 0, E3 0, E4 0 } C_DIS
LIN{ E6POS: X 731.6918, Y -90.6026, Z -172.0150, A 0, B 90, C 0, E1 0, E2 0, E3 0, E4 0 } C_DIS
LIN{ E6POS: X 730.7441, Y -90.2835, Z -172.0150, A 0, B 90, C 0, E1 0, E2 0, E3 0, E4 0 } C_DIS
LIN{ E6POS: X 729.7963, Y -89.9644, Z -172.0150, A 0, B 90, C 0, E1 0, E2 0, E3 0, E4 0 } C_DIS
LIN{ E6POS: X 728.8486, Y -89.6452, Z -172.0150, A 0, B 90, C 0, E1 0, E2 0, E3 0, E4 0 } C_DIS
LIN{ E6POS: X 727.9009, Y -89.3261, Z -172.0150, A 0, B 90, C 0, E1 0, E2 0, E3 0, E4 0 } C_DIS
LIN{ E6POS: X 726.9532, Y -89.0070, Z -172.0150, A 0, B 90, C 0, E1 0, E2 0, E3 0, E4 0 } C_DIS
LIN{ E6POS: X 726.0055, Y -88.6879, Z -172.0150, A 0, B 90, C 0, E1 0, E2 0, E3 0, E4 0 } C_DIS
